LIN {X 0,Y 432.326,Z 417.638,A -85,B 0,C 180,E1 -9497.015,E2 -9497.015} C_VEL
LIN {X 0,Y 432.342,Z 417.631,A -85,B 0,C 180,E1 -9499.819,E2 -9499.819} C_VEL
LIN {X 0,Y 432.316,Z 417.633,A -85,B 0,C 180,E1 -9503.023,E2 -9503.023} C_VEL
LIN {X 0,Y 432.36,Z 417.631,A -85,B 0,C 180,E1 -9505.996,E2 -9505.996} C_VEL
LIN {X 0,Y 432.348,Z 417.629,A -85,B 0,C 180,E1 -9509.49,E2 -9509.49} C_VEL
LIN {X 0,Y 432.394,Z 417.624,A -85,B 0,C 180,E1 -9512.928,E2 -9512.928} C_VEL
LIN {X 0,Y 432.373,Z 417.629,A -85,B 0,C 180,E1 -9516.024,E2 -9516.024} C_VEL
LIN {X 0,Y 432.352,Z 417.628,A -85,B 0,C 180,E1 -9519.046,E2 -9519.046} C_VEL
LIN {X 0,Y 432.38,Z 417.629,A -85,B 0,C 180,E1 -9522.011,E2 -9522.011} C_VEL
LIN {X 0,Y 432.397,Z 417.623,A -85,B 0,C 180,E1 -9524.927,E2 -9524.927} C_VEL
LIN {X 0,Y 432.482,Z 417.615,A -85,B 0,C 180,E1 -9527.804,E2 -9527.804} C_VEL
LIN {X 0,Y 432.465,Z 417.616,A -85,B 0,C 180,E1 -9531.59,E2 -9531.59} C_VEL
LIN {X 0,Y 432.598,Z 417.601,A -85,B 0,C 180,E1 -9534.406,E2 -9534.406} C_VEL
LIN {X 0,Y 432.609,Z 417.6,A -85,B 0,C 180,E1 -9538.138,E2 -9538.138} C_VEL
LIN {X 0,Y 432.735,Z 417.584,A -85,B 0,C 180,E1 -9540,E2 -9540} C_VEL
LIN {X 0,Y 432.594,Z 417.598,A -85,B 0,C 180,E1 -9542.794,E2 -9542.794} C_VEL
LIN {X 0,Y 432.575,Z 417.602,A -85,B 0,C 180,E1 -9546.53,E2 -9546.53} C_VEL
LIN {X 0,Y 432.445,Z 417.618,A -85,B 0,C 180,E1 -9549.353,E2 -9549.353} C_VEL
LIN {X 0,Y 432.432,Z 417.618,A -85,B 0,C 180,E1 -9552.804,E2 -9552.804} C_VEL
LIN {X 0,Y 432.414,Z 417.622,A -85,B 0,C 180,E1 -9556.479,E2 -9556.479} C_VEL
LIN {X 0,Y 432.341,Z 417.633,A -85,B 0,C 180,E1 -9559.961,E2 -9559.961} C_VEL
LIN {X 0,Y 432.322,Z 417.632,A -85,B 0,C 180,E1 -9562.964,E2 -9562.964} C_VEL
LIN {X 0,Y 432.367,Z 417.631,A -85,B 0,C 180,E1 -9566.033,E2 -9566.033} C_VEL
LIN {X 0,Y 432.345,Z 417.629,A -85,B 0,C 180,E1 -9569.188,E2 -9569.188} C_VEL
LIN {X 0,Y 432.325,Z 417.633,A -85,B 0,C 180,E1 -9572.443,E2 -9572.443} C_VEL
LIN {X 0,Y 432.348,Z 417.632,A -85,B 0,C 180,E1 -9575.632,E2 -9575.632} C_VEL
LIN {X 0,Y 432.353,Z 417.628,A -85,B 0,C 180,E1 -9578.716,E2 -9578.716} C_VEL
LIN {X 0,Y 432.338,Z 417.634,A -85,B 0,C 180,E1 -9581.797,E2 -9581.797} C_VEL
LIN {X 0,Y 432.344,Z 417.631,A -85,B 0,C 180,E1 -9584.347,E2 -9584.347} C_VEL
LIN {X 0,Y 432.327,Z 417.632,A -85,B 0,C 180,E1 -9587.015,E2 -9587.015} C_VEL
LIN {X 0,Y 432.34,Z 417.634,A -85,B 0,C 180,E1 -9589.82,E2 -9589.82} C_VEL
LIN {X 0,Y 432.318,Z 417.632,A -85,B 0,C 180,E1 -9593.023,E2 -9593.023} C_VEL
LIN {X 0,Y 432.363,Z 417.63,A -85,B 0,C 180,E1 -9595.997,E2 -9595.997} C_VEL
LIN {X 0,Y 432.399,Z 417.627,A -85,B 0,C 180,E1 -9599.744,E2 -9599.744} C_VEL
LIN {X 0,Y 432.403,Z 417.625,A -85,B 0,C 180,E1 -9603.373,E2 -9603.373} C_VEL
LIN {X 0,Y 432.375,Z 417.629,A -85,B 0,C 180,E1 -9606.024,E2 -9606.024} C_VEL
LIN {X 0,Y 432.355,Z 417.629,A -85,B 0,C 180,E1 -9609.046,E2 -9609.046} C_VEL
LIN {X 0,Y 432.383,Z 417.627,A -85,B 0,C 180,E1 -9612.012,E2 -9612.012} C_VEL
LIN {X 0,Y 432.4,Z 417.626,A -85,B 0,C 180,E1 -9614.927,E2 -9614.927} C_VEL
LIN {X 0,Y 432.461,Z 417.618,A -85,B 0,C 180,E1 -9617.298,E2 -9617.298} C_VEL
LIN {X 0,Y 435.852,Z 429.523,A -85,B 0,C 180,E1 -9618.136,E2 -9618.136} C_VEL
LIN {X 0,Y 436.011,Z 434.479,A -85,B 0,C 180,E1 -9618.494,E2 -9618.494} C_VEL
LIN {X 0,Y 435.45,Z 445.701,A -85,B 0,C 180,E1 -9619.421,E2 -9619.421} C_VEL
LIN {X 0,Y 434.899,Z 455.604,A -85,B 0,C 180,E1 -9620.443,E2 -9620.443} C_VEL
LIN {X 0,Y 434.294,Z 464.879,A -85,B 0,C 180,E1 -9621.626,E2 -9621.626} C_VEL
LIN {X 0,Y 433.884,Z 472.323,A -85,B 0,C 180,E1 -9622.789,E2 -9622.789} C_VEL
LIN {X 0,Y 433.303,Z 479.637,A -85,B 0,C 180,E1 -9624.182,E2 -9624.182} C_VEL
LIN {X 0,Y 432.923,Z 486.364,A -85,B 0,C 180,E1 -9625.811,E2 -9625.811} C_VEL
LIN {X 0,Y 432.607,Z 490.816,A -85,B 0,C 180,E1 -9627.207,E2 -9627.207} C_VEL
LIN {X 0,Y 432.426,Z 493.173,A -85,B 0,C 180,E1 -9628.137,E2 -9628.137} C_VEL
LIN {X 0,Y 432.278,Z 495.194,A -85,B 0,C 180,E1 -9629.127,E2 -9629.127} C_VEL
LIN {X 0,Y 431.525,Z 496.567,A -85,B 0,C 180,E1 -9629.886,E2 -9629.886} C_VEL
LIN {X 0,Y 428.553,Z 498.42,A -85,B 0,C 180,E1 -9631.124,E2 -9631.124} C_VEL
LIN {X 0,Y 426.098,Z 499.436,A -85,B 0,C 180,E1 -9632.129,E2 -9632.129} C_VEL
LIN {X 0,Y 425.064,Z 499.796,A -85,B 0,C 180,E1 -9632.912,E2 -9632.912} C_VEL
LIN {X 0,Y 424.99,Z 499.775,A -85,B 0,C 180,E1 -9633.178,E2 -9633.178} C_VEL
LIN {X 0,Y 425.121,Z 499.284,A -85,B 0,C 180,E1 -9634.742,E2 -9634.742} C_VEL
LIN {X 0,Y 425.3,Z 498.41,A -85,B 0,C 180,E1 -9635.69,E2 -9635.69} C_VEL
LIN {X 0,Y 425.523,Z 495.542,A -85,B 0,C 180,E1 -9637.593,E2 -9637.593} C_VEL
LIN {X 0,Y 425.742,Z 492.253,A -85,B 0,C 180,E1 -9639.023,E2 -9639.023} C_VEL
LIN {X 0,Y 426.172,Z 487.884,A -85,B 0,C 180,E1 -9640.452,E2 -9640.452} C_VEL
LIN {X 0,Y 426.636,Z 481.246,A -85,B 0,C 180,E1 -9642.124,E2 -9642.124} C_VEL
LIN {X 0,Y 427.098,Z 474.255,A -85,B 0,C 180,E1 -9643.516,E2 -9643.516} C_VEL
LIN {X 0,Y 427.766,Z 466.574,A -85,B 0,C 180,E1 -9644.754,E2 -9644.754} C_VEL
LIN {X 0,Y 428.351,Z 457.555,A -85,B 0,C 180,E1 -9645.952,E2 -9645.952} C_VEL
LIN {X 0,Y 428.959,Z 447.467,A -85,B 0,C 180,E1 -9647.03,E2 -9647.03} C_VEL
LIN {X 0,Y 429.566,Z 436.106,A -85,B 0,C 180,E1 -9647.997,E2 -9647.997} C_VEL
LIN {X 0,Y 429.681,Z 432.769,A -85,B 0,C 180,E1 -9648.241,E2 -9648.241} C_VEL
LIN {X 0,Y 426.289,Z 421.626,A -85,B 0,C 180,E1 -9649.115,E2 -9649.115} C_VEL
LIN {X 0,Y 425.389,Z 418.497,A -85,B 0,C 180,E1 -9649.35,E2 -9649.35} C_VEL
LIN {X 0,Y 425.292,Z 418.512,A -85,B 0,C 180,E1 -9652.339,E2 -9652.339} C_VEL
LIN {X 0,Y 425.295,Z 418.504,A -85,B 0,C 180,E1 -9655.446,E2 -9655.446} C_VEL
LIN {X 0,Y 425.353,Z 418.497,A -85,B 0,C 180,E1 -9657.558,E2 -9657.558} C_VEL
LIN {X 0,Y 425.292,Z 418.506,A -85,B 0,C 180,E1 -9660.816,E2 -9660.816} C_VEL
LIN {X 0,Y 425.317,Z 418.508,A -85,B 0,C 180,E1 -9664.288,E2 -9664.288} C_VEL
LIN {X 0,Y 425.284,Z 418.508,A -85,B 0,C 180,E1 -9667.694,E2 -9667.694} C_VEL
LIN {X 0,Y 425.284,Z 418.508,A -85,B 0,C 180,E1 -9670.52,E2 -9670.52} C_VEL
LIN {X 0,Y 425.262,Z 418.509,A -85,B 0,C 180,E1 -9673.351,E2 -9673.351} C_VEL
LIN {X 0,Y 425.263,Z 418.509,A -85,B 0,C 180,E1 -9676.649,E2 -9676.649} C_VEL
LIN {X 0,Y 425.291,Z 418.51,A -85,B 0,C 180,E1 -9679.873,E2 -9679.873} C_VEL
LIN {X 0,Y 425.282,Z 418.508,A -85,B 0,C 180,E1 -9682.488,E2 -9682.488} C_VEL
LIN {X 0,Y 425.312,Z 418.508,A -85,B 0,C 180,E1 -9685.817,E2 -9685.817} C_VEL
LIN {X 0,Y 425.295,Z 418.505,A -85,B 0,C 180,E1 -9689.239,E2 -9689.239} C_VEL
LIN {X 0,Y 425.353,Z 418.498,A -85,B 0,C 180,E1 -9692.442,E2 -9692.442} C_VEL
LIN {X 0,Y 425.352,Z 418.502,A -85,B 0,C 180,E1 -9695.602,E2 -9695.602} C_VEL
LIN {X 0,Y 425.297,Z 418.504,A -85,B 0,C 180,E1 -9698.681,E2 -9698.681} C_VEL
LIN {X 0,Y 425.334,Z 418.507,A -85,B 0,C 180,E1 -9701.703,E2 -9701.703} C_VEL
LIN {X 0,Y 425.352,Z 418.497,A -85,B 0,C 180,E1 -9704.671,E2 -9704.671} C_VEL
LIN {X 0,Y 425.39,Z 418.497,A -85,B 0,C 180,E1 -9705.468,E2 -9705.468} C_VEL
LIN {X 0,Y 428.481,Z 430.294,A -85,B 0,C 180,E1 -9706.336,E2 -9706.336} C_VEL
LIN {X 0,Y 428.042,Z 441.217,A -85,B 0,C 180,E1 -9707.193,E2 -9707.193} C_VEL
LIN {X 0,Y 427.389,Z 452.229,A -85,B 0,C 180,E1 -9708.258,E2 -9708.258} C_VEL
LIN {X 0,Y 427.073,Z 461.189,A -85,B 0,C 180,E1 -9709.331,E2 -9709.331} C_VEL
LIN {X 0,Y 426.483,Z 470.942,A -85,B 0,C 180,E1 -9710.754,E2 -9710.754} C_VEL
LIN {X 0,Y 426.118,Z 478.16,A -85,B 0,C 180,E1 -9712.05,E2 -9712.05} C_VEL
LIN {X 0,Y 425.716,Z 484.179,A -85,B 0,C 180,E1 -9713.364,E2 -9713.364} C_VEL
LIN {X 0,Y 425.501,Z 489.404,A -85,B 0,C 180,E1 -9714.788,E2 -9714.788} C_VEL
LIN {X 0,Y 425.181,Z 493.494,A -85,B 0,C 180,E1 -9716.209,E2 -9716.209} C_VEL
LIN {X 0,Y 425.043,Z 495.618,A -85,B 0,C 180,E1 -9717.157,E2 -9717.157} C_VEL
LIN {X 0,Y 425.115,Z 497.314,A -85,B 0,C 180,E1 -9718.105,E2 -9718.105} C_VEL
LIN {X 0,Y 425.026,Z 498.601,A -85,B 0,C 180,E1 -9719.052,E2 -9719.052} C_VEL
LIN {X 0,Y 425.094,Z 499.904,A -85,B 0,C 180,E1 -9720.947,E2 -9720.947} C_VEL
LIN {X 0,Y 425.168,Z 499.97,A -85,B 0,C 180,E1 -9721.894,E2 -9721.894} C_VEL
LIN {X 0,Y 425.207,Z 498.846,A -85,B 0,C 180,E1 -9723.791,E2 -9723.791} C_VEL
LIN {X 0,Y 425.335,Z 497.69,A -85,B 0,C 180,E1 -9724.739,E2 -9724.739} C_VEL
LIN {X 0,Y 425.688,Z 495.116,A -85,B 0,C 180,E1 -9726.16,E2 -9726.16} C_VEL
LIN {X 0,Y 426.087,Z 490.636,A -85,B 0,C 180,E1 -9727.877,E2 -9727.877} C_VEL
LIN {X 0,Y 426.537,Z 484.964,A -85,B 0,C 180,E1 -9729.484,E2 -9729.484} C_VEL
LIN {X 0,Y 427.038,Z 478.492,A -85,B 0,C 180,E1 -9730.91,E2 -9730.91} C_VEL
LIN {X 0,Y 427.718,Z 470.343,A -85,B 0,C 180,E1 -9732.334,E2 -9732.334} C_VEL
LIN {X 0,Y 428.268,Z 462.012,A -85,B 0,C 180,E1 -9733.524,E2 -9733.524} C_VEL
LIN {X 0,Y 428.866,Z 452.834,A -85,B 0,C 180,E1 -9734.601,E2 -9734.601} C_VEL
LIN {X 0,Y 429.587,Z 441.586,A -85,B 0,C 180,E1 -9735.661,E2 -9735.661} C_VEL
LIN {X 0,Y 429.924,Z 432.512,A -85,B 0,C 180,E1 -9736.362,E2 -9736.362} C_VEL
LIN {X 0,Y 426.422,Z 421.828,A -85,B 0,C 180,E1 -9737.257,E2 -9737.257} C_VEL
LIN {X 0,Y 425.383,Z 418.504,A -85,B 0,C 180,E1 -9737.518,E2 -9737.518} C_VEL
LIN {X 0,Y 425.299,Z 418.517,A -85,B 0,C 180,E1 -9740.305,E2 -9740.305} C_VEL
LIN {X 0,Y 425.308,Z 418.51,A -85,B 0,C 180,E1 -9743.365,E2 -9743.365} C_VEL
LIN {X 0,Y 425.351,Z 418.503,A -85,B 0,C 180,E1 -9746.844,E2 -9746.844} C_VEL
LIN {X 0,Y 425.294,Z 418.509,A -85,B 0,C 180,E1 -9749.719,E2 -9749.719} C_VEL
LIN {X 0,Y 425.285,Z 418.51,A -85,B 0,C 180,E1 -9753.048,E2 -9753.048} C_VEL
LIN {X 0,Y 425.285,Z 418.511,A -85,B 0,C 180,E1 -9755.928,E2 -9755.928} C_VEL
LIN {X 0,Y 425.296,Z 418.508,A -85,B 0,C 180,E1 -9759.042,E2 -9759.042} C_VEL
LIN {X 0,Y 425.278,Z 418.513,A -85,B 0,C 180,E1 -9762.653,E2 -9762.653} C_VEL
LIN {X 0,Y 425.264,Z 418.51,A -85,B 0,C 180,E1 -9766.044,E2 -9766.044} C_VEL
LIN {X 0,Y 425.364,Z 418.669,A -85,B 0,C 180,E1 -9767.585,E2 -9767.585} C_VEL
LIN {X 0,Y 427.208,Z 427.813,A -85,B 0,C 180,E1 -9770.642,E2 -9770.642} C_VEL
LIN {X 0,Y 428.572,Z 435.789,A -85,B 0,C 180,E1 -9773.117,E2 -9773.117} C_VEL
LIN {X 0,Y 427.809,Z 446.144,A -85,B 0,C 180,E1 -9776.044,E2 -9776.044} C_VEL
LIN {X 0,Y 427.039,Z 458.13,A -85,B 0,C 180,E1 -9779.324,E2 -9779.324} C_VEL
LIN {X 0,Y 426.387,Z 470.133,A -85,B 0,C 180,E1 -9782.515,E2 -9782.515} C_VEL
LIN {X 0,Y 425.854,Z 482.082,A -85,B 0,C 180,E1 -9785.633,E2 -9785.633} C_VEL
LIN {X 0,Y 425.349,Z 493.918,A -85,B 0,C 180,E1 -9788.684,E2 -9788.684} C_VEL
LIN {X 0,Y 425.005,Z 505.578,A -85,B 0,C 180,E1 -9791.688,E2 -9791.688} C_VEL
LIN {X 0,Y 424.9,Z 510.092,A -85,B 0,C 180,E1 -9792.85,E2 -9792.85} C_VEL
LIN {X 0,Y 426.68,Z 525.47,A -85,B 0,C 180,E1 -9793.351,E2 -9793.351} C_VEL
LIN {X 0,Y 427.444,Z 538.57,A -85,B 0,C 180,E1 -9793.952,E2 -9793.952} C_VEL
LIN {X 0,Y 427.871,Z 548.142,A -85,B 0,C 180,E1 -9794.519,E2 -9794.519} C_VEL
LIN {X 0,Y 427.109,Z 559.694,A -85,B 0,C 180,E1 -9795.345,E2 -9795.345} C_VEL
LIN {X 0,Y 426.337,Z 571.448,A -85,B 0,C 180,E1 -9796.414,E2 -9796.414} C_VEL
LIN {X 0,Y 425.858,Z 580.24,A -85,B 0,C 180,E1 -9797.401,E2 -9797.401} C_VEL
LIN {X 0,Y 425.303,Z 588.867,A -85,B 0,C 180,E1 -9798.562,E2 -9798.562} C_VEL
LIN {X 0,Y 424.829,Z 597.558,A -85,B 0,C 180,E1 -9799.997,E2 -9799.997} C_VEL
LIN {X 0,Y 424.634,Z 604.578,A -85,B 0,C 180,E1 -9801.433,E2 -9801.433} C_VEL
LIN {X 0,Y 424.578,Z 610.395,A -85,B 0,C 180,E1 -9802.916,E2 -9802.916} C_VEL
LIN {X 0,Y 424.589,Z 614.669,A -85,B 0,C 180,E1 -9804.3,E2 -9804.3} C_VEL
LIN {X 0,Y 424.686,Z 617.04,A -85,B 0,C 180,E1 -9805.253,E2 -9805.253} C_VEL
LIN {X 0,Y 424.718,Z 618.941,A -85,B 0,C 180,E1 -9806.205,E2 -9806.205} C_VEL
LIN {X 0,Y 424.7,Z 620.365,A -85,B 0,C 180,E1 -9807.154,E2 -9807.154} C_VEL
LIN {X 0,Y 424.921,Z 622.033,A -85,B 0,C 180,E1 -9809.052,E2 -9809.052} C_VEL
LIN {X 0,Y 424.922,Z 622.232,A -85,B 0,C 180,E1 -9810,E2 -9810} C_VEL
LIN {X 0,Y 424.922,Z 621.99,A -85,B 0,C 180,E1 -9810.947,E2 -9810.947} C_VEL
LIN {X 0,Y 424.71,Z 620.274,A -85,B 0,C 180,E1 -9812.845,E2 -9812.845} C_VEL
LIN {X 0,Y 424.715,Z 618.797,A -85,B 0,C 180,E1 -9813.795,E2 -9813.795} C_VEL
LIN {X 0,Y 424.651,Z 615.717,A -85,B 0,C 180,E1 -9815.222,E2 -9815.222} C_VEL
LIN {X 0,Y 424.582,Z 611.387,A -85,B 0,C 180,E1 -9816.702,E2 -9816.702} C_VEL
LIN {X 0,Y 424.656,Z 605.163,A -85,B 0,C 180,E1 -9818.326,E2 -9818.326} C_VEL
LIN {X 0,Y 424.83,Z 598.22,A -85,B 0,C 180,E1 -9819.762,E2 -9819.762} C_VEL
LIN {X 0,Y 425.196,Z 589.631,A -85,B 0,C 180,E1 -9821.199,E2 -9821.199} C_VEL
LIN {X 0,Y 425.761,Z 580.824,A -85,B 0,C 180,E1 -9822.391,E2 -9822.391} C_VEL
LIN {X 0,Y 426.226,Z 571.171,A -85,B 0,C 180,E1 -9823.468,E2 -9823.468} C_VEL
LIN {X 0,Y 426.938,Z 559.25,A -85,B 0,C 180,E1 -9824.539,E2 -9824.539} C_VEL
LIN {X 0,Y 427.689,Z 547.375,A -85,B 0,C 180,E1 -9825.365,E2 -9825.365} C_VEL
LIN {X 0,Y 427.38,Z 540.977,A -85,B 0,C 180,E1 -9825.743,E2 -9825.743} C_VEL
LIN {X 0,Y 426.502,Z 527.164,A -85,B 0,C 180,E1 -9826.399,E2 -9826.399} C_VEL
LIN {X 0,Y 425.159,Z 513.732,A -85,B 0,C 180,E1 -9826.84,E2 -9826.84} C_VEL
LIN {X 0,Y 424.856,Z 510.351,A -85,B 0,C 180,E1 -9826.941,E2 -9826.941} C_VEL
LIN {X 0,Y 425.219,Z 497.119,A -85,B 0,C 180,E1 -9830.309,E2 -9830.309} C_VEL
LIN {X 0,Y 425.617,Z 485.211,A -85,B 0,C 180,E1 -9833.347,E2 -9833.347} C_VEL
LIN {X 0,Y 426.117,Z 473.121,A -85,B 0,C 180,E1 -9836.443,E2 -9836.443} C_VEL
LIN {X 0,Y 426.832,Z 458.896,A -85,B 0,C 180,E1 -9840.145,E2 -9840.145} C_VEL
LIN {X 0,Y 427.475,Z 446.582,A -85,B 0,C 180,E1 -9843.438,E2 -9843.438} C_VEL
LIN {X 0,Y 428.244,Z 435.561,A -85,B 0,C 180,E1 -9846.472,E2 -9846.472} C_VEL
LIN {X 0,Y 427.7,Z 430.625,A -85,B 0,C 180,E1 -9847.932,E2 -9847.932} C_VEL
LIN {X 0,Y 425.77,Z 420.667,A -85,B 0,C 180,E1 -9851.058,E2 -9851.058} C_VEL
LIN {X 0,Y 425.335,Z 418.505,A -85,B 0,C 180,E1 -9851.768,E2 -9851.768} C_VEL
LIN {X 0,Y 425.29,Z 418.513,A -85,B 0,C 180,E1 -9855.282,E2 -9855.282} C_VEL
LIN {X 0,Y 425.277,Z 418.512,A -85,B 0,C 180,E1 -9858.622,E2 -9858.622} C_VEL
LIN {X 0,Y 425.317,Z 418.505,A -85,B 0,C 180,E1 -9861.103,E2 -9861.103} C_VEL
LIN {X 0,Y 425.301,Z 418.508,A -85,B 0,C 180,E1 -9864.664,E2 -9864.664} C_VEL
LIN {X 0,Y 425.266,Z 418.515,A -85,B 0,C 180,E1 -9868.073,E2 -9868.073} C_VEL
LIN {X 0,Y 425.332,Z 418.503,A -85,B 0,C 180,E1 -9871.368,E2 -9871.368} C_VEL
LIN {X 0,Y 425.297,Z 418.509,A -85,B 0,C 180,E1 -9874.555,E2 -9874.555} C_VEL
LIN {X 0,Y 425.289,Z 418.51,A -85,B 0,C 180,E1 -9877.661,E2 -9877.661} C_VEL
LIN {X 0,Y 425.363,Z 418.5,A -85,B 0,C 180,E1 -9880.704,E2 -9880.704} C_VEL
LIN {X 0,Y 425.39,Z 418.497,A -85,B 0,C 180,E1 -9883.688,E2 -9883.688} C_VEL
LIN {X 0,Y 425.431,Z 418.492,A -85,B 0,C 180,E1 -9887.599,E2 -9887.599} C_VEL
LIN {X 0,Y 425.41,Z 418.493,A -85,B 0,C 180,E1 -9891.449,E2 -9891.449} C_VEL
LIN {X 0,Y 425.554,Z 418.479,A -85,B 0,C 180,E1 -9894.313,E2 -9894.313} C_VEL
LIN {X 0,Y 425.578,Z 418.476,A -85,B 0,C 180,E1 -9898.107,E2 -9898.107} C_VEL
LIN {X 0,Y 425.705,Z 418.46,A -85,B 0,C 180,E1 -9900,E2 -9900} C_VEL
LIN {X 0,Y 425.547,Z 418.475,A -85,B 0,C 180,E1 -9902.84,E2 -9902.84} C_VEL
LIN {X 0,Y 425.532,Z 418.478,A -85,B 0,C 180,E1 -9906.649,E2 -9906.649} C_VEL
LIN {X 0,Y 425.403,Z 418.496,A -85,B 0,C 180,E1 -9909.51,E2 -9909.51} C_VEL
LIN {X 0,Y 425.395,Z 418.495,A -85,B 0,C 180,E1 -9912.904,E2 -9912.904} C_VEL
LIN {X 0,Y 425.363,Z 418.499,A -85,B 0,C 180,E1 -9916.605,E2 -9916.605} C_VEL
LIN {X 0,Y 425.331,Z 418.505,A -85,B 0,C 180,E1 -9919.636,E2 -9919.636} C_VEL
LIN {X 0,Y 425.309,Z 418.507,A -85,B 0,C 180,E1 -9923.365,E2 -9923.365} C_VEL
LIN {X 0,Y 425.35,Z 418.5,A -85,B 0,C 180,E1 -9926.845,E2 -9926.845} C_VEL
LIN {X 0,Y 425.293,Z 418.512,A -85,B 0,C 180,E1 -9929.72,E2 -9929.72} C_VEL
LIN {X 0,Y 425.284,Z 418.509,A -85,B 0,C 180,E1 -9933.048,E2 -9933.048} C_VEL
LIN {X 0,Y 425.287,Z 418.513,A -85,B 0,C 180,E1 -9935.929,E2 -9935.929} C_VEL
LIN {X 0,Y 425.302,Z 418.506,A -85,B 0,C 180,E1 -9939.044,E2 -9939.044} C_VEL
LIN {X 0,Y 425.28,Z 418.509,A -85,B 0,C 180,E1 -9942.653,E2 -9942.653} C_VEL
LIN {X 0,Y 425.271,Z 418.513,A -85,B 0,C 180,E1 -9946.045,E2 -9946.045} C_VEL
LIN {X 0,Y 425.278,Z 418.509,A -85,B 0,C 180,E1 -9948.622,E2 -9948.622} C_VEL
LIN {X 0,Y 425.316,Z 418.505,A -85,B 0,C 180,E1 -9951.103,E2 -9951.103} C_VEL
LIN {X 0,Y 425.303,Z 418.506,A -85,B 0,C 180,E1 -9954.665,E2 -9954.665} C_VEL
LIN {X 0,Y 425.276,Z 418.513,A -85,B 0,C 180,E1 -9958.074,E2 -9958.074} C_VEL
LIN {X 0,Y 425.341,Z 418.505,A -85,B 0,C 180,E1 -9961.369,E2 -9961.369} C_VEL
LIN {X 0,Y 425.299,Z 418.506,A -85,B 0,C 180,E1 -9964.555,E2 -9964.555} C_VEL
LIN {X 0,Y 425.291,Z 418.512,A -85,B 0,C 180,E1 -9967.662,E2 -9967.662} C_VEL
LIN {X 0,Y 425.366,Z 418.498,A -85,B 0,C 180,E1 -9970.704,E2 -9970.704} C_VEL
LIN {X 0,Y 425.393,Z 418.499,A -85,B 0,C 180,E1 -9973.689,E2 -9973.689} C_VEL
LIN {X 0,Y 425.401,Z 418.497,A -85,B 0,C 180,E1 -9977.032,E2 -9977.032} C_VEL
LIN {X 0,Y 429.015,Z 431.02,A -85,B 0,C 180,E1 -9977.944,E2 -9977.944} C_VEL
LIN {X 0,Y 429.174,Z 435.923,A -85,B 0,C 180,E1 -9978.308,E2 -9978.308} C_VEL
LIN {X 0,Y 428.604,Z 447.061,A -85,B 0,C 180,E1 -9979.25,E2 -9979.25} C_VEL
LIN {X 0,Y 428.016,Z 456.896,A -85,B 0,C 180,E1 -9980.287,E2 -9980.287} C_VEL
LIN {X 0,Y 427.377,Z 466.112,A -85,B 0,C 180,E1 -9981.489,E2 -9981.489} C_VEL
LIN {X 0,Y 426.942,Z 473.519,A -85,B 0,C 180,E1 -9982.671,E2 -9982.671} C_VEL
LIN {X 0,Y 426.338,Z 480.801,A -85,B 0,C 180,E1 -9984.087,E2 -9984.087} C_VEL
LIN {X 0,Y 425.934,Z 487.494,A -85,B 0,C 180,E1 -9985.742,E2 -9985.742} C_VEL
LIN {X 0,Y 425.603,Z 491.92,A -85,B 0,C 180,E1 -9987.161,E2 -9987.161} C_VEL
LIN {X 0,Y 425.417,Z 494.257,A -85,B 0,C 180,E1 -9988.107,E2 -9988.107} C_VEL
LIN {X 0,Y 425.194,Z 497.682,A -85,B 0,C 180,E1 -9990,E2 -9990} C_VEL
LIN {X 0,Y 425.026,Z 498.79,A -85,B 0,C 180,E1 -9990.948,E2 -9990.948} C_VEL
LIN {X 0,Y 425.097,Z 499.462,A -85,B 0,C 180,E1 -9991.895,E2 -9991.895} C_VEL
LIN {X 0,Y 424.99,Z 499.775,A -85,B 0,C 180,E1 -9993.178,E2 -9993.178} C_VEL
LIN {X 0,Y 424.374,Z 499.785,A -85,B 0,C 180,E1 -9993.971,E2 -9993.971} C_VEL
LIN {X 0,Y 421.648,Z 499.39,A -85,B 0,C 180,E1 -9995.263,E2 -9995.263} C_VEL
LIN {X 0,Y 418.977,Z 498.335,A -85,B 0,C 180,E1 -9996.561,E2 -9996.561} C_VEL
LIN {X 0,Y 418.459,Z 497.119,A -85,B 0,C 180,E1 -9997.353,E2 -9997.353} C_VEL
LIN {X 0,Y 418.795,Z 493.18,A -85,B 0,C 180,E1 -9999.174,E2 -9999.174} C_VEL
LIN {X 0,Y 419.251,Z 488.785,A -85,B 0,C 180,E1 -10000.626,E2 -10000.626} C_VEL
LIN {X 0,Y 419.738,Z 482.107,A -85,B 0,C 180,E1 -10002.327,E2 -10002.327} C_VEL
LIN {X 0,Y 420.243,Z 475.129,A -85,B 0,C 180,E1 -10003.732,E2 -10003.732} C_VEL
LIN {X 0,Y 420.959,Z 467.363,A -85,B 0,C 180,E1 -10004.998,E2 -10004.998} C_VEL
LIN {X 0,Y 421.552,Z 458.292,A -85,B 0,C 180,E1 -10006.216,E2 -10006.216} C_VEL
LIN {X 0,Y 422.205,Z 448.128,A -85,B 0,C 180,E1 -10007.311,E2 -10007.311} C_VEL
LIN {X 0,Y 422.843,Z 436.401,A -85,B 0,C 180,E1 -10008.316,E2 -10008.316} C_VEL
LIN {X 0,Y 422.588,Z 433.25,A -85,B 0,C 180,E1 -10008.564,E2 -10008.564} C_VEL
LIN {X 0,Y 419.259,Z 422.462,A -85,B 0,C 180,E1 -10009.425,E2 -10009.425} C_VEL
LIN {X 0,Y 418.312,Z 419.38,A -85,B 0,C 180,E1 -10009.671,E2 -10009.671} C_VEL
LIN {X 0,Y 418.236,Z 419.386,A -85,B 0,C 180,E1 -10012.737,E2 -10012.737} C_VEL
LIN {X 0,Y 418.272,Z 419.382,A -85,B 0,C 180,E1 -10015.904,E2 -10015.904} C_VEL
LIN {X 0,Y 418.269,Z 419.379,A -85,B 0,C 180,E1 -10019.162,E2 -10019.162} C_VEL
LIN {X 0,Y 418.262,Z 419.381,A -85,B 0,C 180,E1 -10022.844,E2 -10022.844} C_VEL
LIN {X 0,Y 418.25,Z 419.389,A -85,B 0,C 180,E1 -10026.238,E2 -10026.238} C_VEL
LIN {X 0,Y 418.253,Z 419.384,A -85,B 0,C 180,E1 -10029.682,E2 -10029.682} C_VEL
LIN {X 0,Y 418.234,Z 419.388,A -85,B 0,C 180,E1 -10032.321,E2 -10032.321} C_VEL
LIN {X 0,Y 418.242,Z 419.383,A -85,B 0,C 180,E1 -10035.109,E2 -10035.109} C_VEL
LIN {X 0,Y 418.245,Z 419.387,A -85,B 0,C 180,E1 -10037.767,E2 -10037.767} C_VEL
LIN {X 0,Y 418.257,Z 419.382,A -85,B 0,C 180,E1 -10040.619,E2 -10040.619} C_VEL
LIN {X 0,Y 418.248,Z 419.389,A -85,B 0,C 180,E1 -10043.976,E2 -10043.976} C_VEL
LIN {X 0,Y 418.262,Z 419.381,A -85,B 0,C 180,E1 -10047.156,E2 -10047.156} C_VEL
LIN {X 0,Y 418.273,Z 419.379,A -85,B 0,C 180,E1 -10050.895,E2 -10050.895} C_VEL
LIN {X 0,Y 418.272,Z 419.383,A -85,B 0,C 180,E1 -10054.096,E2 -10054.096} C_VEL
LIN {X 0,Y 418.236,Z 419.385,A -85,B 0,C 180,E1 -10057.263,E2 -10057.263} C_VEL
LIN {X 0,Y 418.287,Z 419.378,A -85,B 0,C 180,E1 -10060.364,E2 -10060.364} C_VEL
LIN {X 0,Y 418.321,Z 419.377,A -85,B 0,C 180,E1 -10063.405,E2 -10063.405} C_VEL
LIN {X 0,Y 418.352,Z 419.469,A -85,B 0,C 180,E1 -10065.28,E2 -10065.28} C_VEL
LIN {X 0,Y 421.505,Z 431.457,A -85,B 0,C 180,E1 -10066.168,E2 -10066.168} C_VEL
LIN {X 0,Y 421.057,Z 443.001,A -85,B 0,C 180,E1 -10067.1,E2 -10067.1} C_VEL
LIN {X 0,Y 420.413,Z 453.841,A -85,B 0,C 180,E1 -10068.183,E2 -10068.183} C_VEL
LIN {X 0,Y 420.022,Z 463.566,A -85,B 0,C 180,E1 -10069.394,E2 -10069.394} C_VEL
LIN {X 0,Y 419.45,Z 473.098,A -85,B 0,C 180,E1 -10070.841,E2 -10070.841} C_VEL
LIN {X 0,Y 419.033,Z 480.704,A -85,B 0,C 180,E1 -10072.289,E2 -10072.289} C_VEL
LIN {X 0,Y 418.636,Z 486.865,A -85,B 0,C 180,E1 -10073.735,E2 -10073.735} C_VEL
LIN {X 0,Y 418.281,Z 491.774,A -85,B 0,C 180,E1 -10075.181,E2 -10075.181} C_VEL
LIN {X 0,Y 418.176,Z 495.538,A -85,B 0,C 180,E1 -10076.628,E2 -10076.628} C_VEL
LIN {X 0,Y 418.093,Z 498.285,A -85,B 0,C 180,E1 -10078.073,E2 -10078.073} C_VEL
LIN {X 0,Y 418.004,Z 499.603,A -85,B 0,C 180,E1 -10079.036,E2 -10079.036} C_VEL
LIN {X 0,Y 418.092,Z 500.947,A -85,B 0,C 180,E1 -10080.963,E2 -10080.963} C_VEL
LIN {X 0,Y 418.172,Z 501.042,A -85,B 0,C 180,E1 -10081.926,E2 -10081.926} C_VEL
LIN {X 0,Y 418.183,Z 500.705,A -85,B 0,C 180,E1 -10082.89,E2 -10082.89} C_VEL
LIN {X 0,Y 418.352,Z 498.848,A -85,B 0,C 180,E1 -10084.818,E2 -10084.818} C_VEL
LIN {X 0,Y 418.74,Z 496.304,A -85,B 0,C 180,E1 -10086.263,E2 -10086.263} C_VEL
LIN {X 0,Y 419.103,Z 492.756,A -85,B 0,C 180,E1 -10087.71,E2 -10087.71} C_VEL
LIN {X 0,Y 419.482,Z 488.079,A -85,B 0,C 180,E1 -10089.158,E2 -10089.158} C_VEL
LIN {X 0,Y 420.046,Z 480.96,A -85,B 0,C 180,E1 -10090.849,E2 -10090.849} C_VEL
LIN {X 0,Y 420.742,Z 473.242,A -85,B 0,C 180,E1 -10092.297,E2 -10092.297} C_VEL
LIN {X 0,Y 421.513,Z 463.526,A -85,B 0,C 180,E1 -10093.745,E2 -10093.745} C_VEL
LIN {X 0,Y 422.165,Z 454.459,A -85,B 0,C 180,E1 -10094.838,E2 -10094.838} C_VEL
LIN {X 0,Y 422.944,Z 443.313,A -85,B 0,C 180,E1 -10095.913,E2 -10095.913} C_VEL
LIN {X 0,Y 423.32,Z 434.494,A -85,B 0,C 180,E1 -10096.615,E2 -10096.615} C_VEL
LIN {X 0,Y 419.956,Z 424.093,A -85,B 0,C 180,E1 -10097.532,E2 -10097.532} C_VEL
LIN {X 0,Y 418.32,Z 419.386,A -85,B 0,C 180,E1 -10097.918,E2 -10097.918} C_VEL
LIN {X 0,Y 418.254,Z 419.393,A -85,B 0,C 180,E1 -10100.663,E2 -10100.663} C_VEL
LIN {X 0,Y 418.289,Z 419.384,A -85,B 0,C 180,E1 -10103.781,E2 -10103.781} C_VEL
LIN {X 0,Y 418.313,Z 419.381,A -85,B 0,C 180,E1 -10107.07,E2 -10107.07} C_VEL
LIN {X 0,Y 418.248,Z 419.388,A -85,B 0,C 180,E1 -10110.272,E2 -10110.272} C_VEL
LIN {X 0,Y 418.252,Z 419.384,A -85,B 0,C 180,E1 -10113.677,E2 -10113.677} C_VEL
LIN {X 0,Y 418.243,Z 419.386,A -85,B 0,C 180,E1 -10117.224,E2 -10117.224} C_VEL
LIN {X 0,Y 418.252,Z 419.386,A -85,B 0,C 180,E1 -10119.682,E2 -10119.682} C_VEL
LIN {X 0,Y 418.233,Z 419.387,A -85,B 0,C 180,E1 -10122.321,E2 -10122.321} C_VEL
LIN {X 0,Y 418.239,Z 419.392,A -85,B 0,C 180,E1 -10125.109,E2 -10125.109} C_VEL
LIN {X 0,Y 418.281,Z 419.414,A -85,B 0,C 180,E1 -10127.176,E2 -10127.176} C_VEL
LIN {X 0,Y 420.304,Z 429.337,A -85,B 0,C 180,E1 -10130.549,E2 -10130.549} C_VEL
LIN {X 0,Y 421.572,Z 436.433,A -85,B 0,C 180,E1 -10132.82,E2 -10132.82} C_VEL
LIN {X 0,Y 421.307,Z 441.408,A -85,B 0,C 180,E1 -10134.278,E2 -10134.278} C_VEL
LIN {X 0,Y 420.417,Z 453.36,A -85,B 0,C 180,E1 -10137.66,E2 -10137.66} C_VEL
LIN {X 0,Y 419.68,Z 465.323,A -85,B 0,C 180,E1 -10140.945,E2 -10140.945} C_VEL
LIN {X 0,Y 418.956,Z 478.963,A -85,B 0,C 180,E1 -10144.601,E2 -10144.601} C_VEL
LIN {X 0,Y 418.416,Z 491.422,A -85,B 0,C 180,E1 -10147.891,E2 -10147.891} C_VEL
LIN {X 0,Y 417.955,Z 504.601,A -85,B 0,C 180,E1 -10151.368,E2 -10151.368} C_VEL
LIN {X 0,Y 417.835,Z 509.039,A -85,B 0,C 180,E1 -10152.531,E2 -10152.531} C_VEL
LIN {X 0,Y 419.633,Z 524.36,A -85,B 0,C 180,E1 -10153.042,E2 -10153.042} C_VEL
LIN {X 0,Y 420.484,Z 537.86,A -85,B 0,C 180,E1 -10153.679,E2 -10153.679} C_VEL
LIN {X 0,Y 420.982,Z 547.376,A -85,B 0,C 180,E1 -10154.259,E2 -10154.259} C_VEL
LIN {X 0,Y 420.198,Z 558.868,A -85,B 0,C 180,E1 -10155.099,E2 -10155.099} C_VEL
LIN {X 0,Y 419.378,Z 570.578,A -85,B 0,C 180,E1 -10156.184,E2 -10156.184} C_VEL
LIN {X 0,Y 418.841,Z 579.616,A -85,B 0,C 180,E1 -10157.221,E2 -10157.221} C_VEL
LIN {X 0,Y 418.27,Z 587.945,A -85,B 0,C 180,E1 -10158.367,E2 -10158.367} C_VEL
LIN {X 0,Y 417.762,Z 596.607,A -85,B 0,C 180,E1 -10159.826,E2 -10159.826} C_VEL
LIN {X 0,Y 417.558,Z 603.614,A -85,B 0,C 180,E1 -10161.287,E2 -10161.287} C_VEL
LIN {X 0,Y 417.497,Z 609.252,A -85,B 0,C 180,E1 -10162.747,E2 -10162.747} C_VEL
LIN {X 0,Y 417.535,Z 613.688,A -85,B 0,C 180,E1 -10164.203,E2 -10164.203} C_VEL
LIN {X 0,Y 417.638,Z 616.055,A -85,B 0,C 180,E1 -10165.173,E2 -10165.173} C_VEL
LIN {X 0,Y 417.68,Z 617.947,A -85,B 0,C 180,E1 -10166.141,E2 -10166.141} C_VEL
LIN {X 0,Y 417.657,Z 619.366,A -85,B 0,C 180,E1 -10167.106,E2 -10167.106} C_VEL
LIN {X 0,Y 417.897,Z 621.028,A -85,B 0,C 180,E1 -10169.036,E2 -10169.036} C_VEL
LIN {X 0,Y 417.902,Z 621.218,A -85,B 0,C 180,E1 -10170,E2 -10170} C_VEL
LIN {X 0,Y 417.898,Z 620.971,A -85,B 0,C 180,E1 -10170.963,E2 -10170.963} C_VEL
LIN {X 0,Y 417.669,Z 619.241,A -85,B 0,C 180,E1 -10172.893,E2 -10172.893} C_VEL
LIN {X 0,Y 417.677,Z 617.753,A -85,B 0,C 180,E1 -10173.859,E2 -10173.859} C_VEL
LIN {X 0,Y 417.587,Z 614.658,A -85,B 0,C 180,E1 -10175.311,E2 -10175.311} C_VEL
LIN {X 0,Y 417.519,Z 610.476,A -85,B 0,C 180,E1 -10176.767,E2 -10176.767} C_VEL
LIN {X 0,Y 417.586,Z 604.067,A -85,B 0,C 180,E1 -10178.468,E2 -10178.468} C_VEL
LIN {X 0,Y 417.778,Z 597.106,A -85,B 0,C 180,E1 -10179.929,E2 -10179.929} C_VEL
LIN {X 0,Y 418.179,Z 588.492,A -85,B 0,C 180,E1 -10181.389,E2 -10181.389} C_VEL
LIN {X 0,Y 418.793,Z 579.662,A -85,B 0,C 180,E1 -10182.601,E2 -10182.601} C_VEL
LIN {X 0,Y 418.986,Z 573.052,A -85,B 0,C 180,E1 -10183.373,E2 -10183.373} C_VEL
LIN {X 0,Y 419.756,Z 562.354,A -85,B 0,C 180,E1 -10184.421,E2 -10184.421} C_VEL
LIN {X 0,Y 420.462,Z 551.567,A -85,B 0,C 180,E1 -10185.263,E2 -10185.263} C_VEL
LIN {X 0,Y 420.688,Z 545.022,A -85,B 0,C 180,E1 -10185.69,E2 -10185.69} C_VEL
LIN {X 0,Y 419.993,Z 534.664,A -85,B 0,C 180,E1 -10186.277,E2 -10186.277} C_VEL
LIN {X 0,Y 419.012,Z 521.336,A -85,B 0,C 180,E1 -10186.844,E2 -10186.844} C_VEL
LIN {X 0,Y 417.783,Z 509.362,A -85,B 0,C 180,E1 -10187.205,E2 -10187.205} C_VEL
LIN {X 0,Y 418.158,Z 496.065,A -85,B 0,C 180,E1 -10190.668,E2 -10190.668} C_VEL
LIN {X 0,Y 418.648,Z 483.195,A -85,B 0,C 180,E1 -10194.022,E2 -10194.022} C_VEL
LIN {X 0,Y 419.187,Z 470.681,A -85,B 0,C 180,E1 -10197.304,E2 -10197.304} C_VEL
LIN {X 0,Y 419.895,Z 457.951,A -85,B 0,C 180,E1 -10200.697,E2 -10200.697} C_VEL
LIN {X 0,Y 420.698,Z 444.727,A -85,B 0,C 180,E1 -10204.32,E2 -10204.32} C_VEL
LIN {X 0,Y 421.264,Z 435.571,A -85,B 0,C 180,E1 -10206.912,E2 -10206.912} C_VEL
LIN {X 0,Y 419.784,Z 426.792,A -85,B 0,C 180,E1 -10209.634,E2 -10209.634} C_VEL
LIN {X 0,Y 418.28,Z 419.383,A -85,B 0,C 180,E1 -10212.097,E2 -10212.097} C_VEL
LIN {X 0,Y 418.24,Z 419.392,A -85,B 0,C 180,E1 -10215.109,E2 -10215.109} C_VEL
LIN {X 0,Y 418.243,Z 419.387,A -85,B 0,C 180,E1 -10217.767,E2 -10217.767} C_VEL
LIN {X 0,Y 418.261,Z 419.386,A -85,B 0,C 180,E1 -10220.618,E2 -10220.618} C_VEL
LIN {X 0,Y 418.247,Z 419.389,A -85,B 0,C 180,E1 -10223.976,E2 -10223.976} C_VEL
LIN {X 0,Y 418.258,Z 419.383,A -85,B 0,C 180,E1 -10227.156,E2 -10227.156} C_VEL
LIN {X 0,Y 418.269,Z 419.383,A -85,B 0,C 180,E1 -10230.895,E2 -10230.895} C_VEL
LIN {X 0,Y 418.272,Z 419.386,A -85,B 0,C 180,E1 -10234.096,E2 -10234.096} C_VEL
LIN {X 0,Y 418.239,Z 419.386,A -85,B 0,C 180,E1 -10237.264,E2 -10237.264} C_VEL
LIN {X 0,Y 418.285,Z 419.384,A -85,B 0,C 180,E1 -10240.364,E2 -10240.364} C_VEL
LIN {X 0,Y 418.318,Z 419.376,A -85,B 0,C 180,E1 -10243.405,E2 -10243.405} C_VEL
LIN {X 0,Y 418.356,Z 419.371,A -85,B 0,C 180,E1 -10246.994,E2 -10246.994} C_VEL
LIN {X 0,Y 418.359,Z 419.374,A -85,B 0,C 180,E1 -10250.329,E2 -10250.329} C_VEL
LIN {X 0,Y 418.481,Z 419.355,A -85,B 0,C 180,E1 -10253.249,E2 -10253.249} C_VEL
LIN {X 0,Y 418.344,Z 419.373,A -85,B 0,C 180,E1 -10255.182,E2 -10255.182} C_VEL
LIN {X 0,Y 418.547,Z 419.352,A -85,B 0,C 180,E1 -10258.076,E2 -10258.076} C_VEL
LIN {X 0,Y 418.675,Z 419.336,A -85,B 0,C 180,E1 -10260,E2 -10260} C_VEL
LIN {X 0,Y 418.502,Z 419.353,A -85,B 0,C 180,E1 -10262.888,E2 -10262.888} C_VEL
LIN {X 0,Y 418.495,Z 419.354,A -85,B 0,C 180,E1 -10266.751,E2 -10266.751} C_VEL
LIN {X 0,Y 418.343,Z 419.376,A -85,B 0,C 180,E1 -10269.672,E2 -10269.672} C_VEL
LIN {X 0,Y 418.348,Z 419.372,A -85,B 0,C 180,E1 -10273.001,E2 -10273.001} C_VEL
LIN {X 0,Y 418.315,Z 419.376,A -85,B 0,C 180,E1 -10276.736,E2 -10276.736} C_VEL
LIN {X 0,Y 418.273,Z 419.386,A -85,B 0,C 180,E1 -10279.791,E2 -10279.791} C_VEL
LIN {X 0,Y 418.24,Z 419.386,A -85,B 0,C 180,E1 -10282.736,E2 -10282.736} C_VEL
LIN {X 0,Y 418.273,Z 419.386,A -85,B 0,C 180,E1 -10285.904,E2 -10285.904} C_VEL
LIN {X 0,Y 418.267,Z 419.382,A -85,B 0,C 180,E1 -10289.162,E2 -10289.162} C_VEL
LIN {X 0,Y 418.259,Z 419.383,A -85,B 0,C 180,E1 -10292.844,E2 -10292.844} C_VEL
LIN {X 0,Y 418.251,Z 419.387,A -85,B 0,C 180,E1 -10296.239,E2 -10296.239} C_VEL
LIN {X 0,Y 418.255,Z 419.388,A -85,B 0,C 180,E1 -10299.682,E2 -10299.682} C_VEL
LIN {X 0,Y 418.234,Z 419.388,A -85,B 0,C 180,E1 -10302.322,E2 -10302.322} C_VEL
LIN {X 0,Y 418.245,Z 419.386,A -85,B 0,C 180,E1 -10305.11,E2 -10305.11} C_VEL
LIN {X 0,Y 418.245,Z 419.39,A -85,B 0,C 180,E1 -10307.767,E2 -10307.767} C_VEL
LIN {X 0,Y 418.26,Z 419.383,A -85,B 0,C 180,E1 -10310.619,E2 -10310.619} C_VEL
LIN {X 0,Y 418.249,Z 419.389,A -85,B 0,C 180,E1 -10313.977,E2 -10313.977} C_VEL
LIN {X 0,Y 418.263,Z 419.384,A -85,B 0,C 180,E1 -10317.156,E2 -10317.156} C_VEL
LIN {X 0,Y 418.278,Z 419.381,A -85,B 0,C 180,E1 -10320.839,E2 -10320.839} C_VEL
LIN {X 0,Y 418.274,Z 419.384,A -85,B 0,C 180,E1 -10324.096,E2 -10324.096} C_VEL
LIN {X 0,Y 418.242,Z 419.387,A -85,B 0,C 180,E1 -10327.264,E2 -10327.264} C_VEL
LIN {X 0,Y 418.287,Z 419.381,A -85,B 0,C 180,E1 -10330.365,E2 -10330.365} C_VEL
LIN {X 0,Y 418.321,Z 419.379,A -85,B 0,C 180,E1 -10333.405,E2 -10333.405} C_VEL
LIN {X 0,Y 418.355,Z 419.486,A -85,B 0,C 180,E1 -10336.781,E2 -10336.781} C_VEL
LIN {X 0,Y 421.734,Z 430.889,A -85,B 0,C 180,E1 -10337.611,E2 -10337.611} C_VEL
LIN {X 0,Y 422.441,Z 434.172,A -85,B 0,C 180,E1 -10337.876,E2 -10337.876} C_VEL
LIN {X 0,Y 421.868,Z 445.895,A -85,B 0,C 180,E1 -10338.833,E2 -10338.833} C_VEL
LIN {X 0,Y 421.255,Z 456.39,A -85,B 0,C 180,E1 -10339.921,E2 -10339.921} C_VEL
LIN {X 0,Y 420.574,Z 465.758,A -85,B 0,C 180,E1 -10341.116,E2 -10341.116} C_VEL
LIN {X 0,Y 420.016,Z 473.38,A -85,B 0,C 180,E1 -10342.307,E2 -10342.307} C_VEL
LIN {X 0,Y 419.517,Z 480.866,A -85,B 0,C 180,E1 -10343.749,E2 -10343.749} C_VEL
LIN {X 0,Y 419.046,Z 486.879,A -85,B 0,C 180,E1 -10345.19,E2 -10345.19} C_VEL
LIN {X 0,Y 418.671,Z 491.655,A -85,B 0,C 180,E1 -10346.632,E2 -10346.632} C_VEL
LIN {X 0,Y 418.406,Z 495.34,A -85,B 0,C 180,E1 -10348.075,E2 -10348.075} C_VEL
LIN {X 0,Y 418.175,Z 498.742,A -85,B 0,C 180,E1 -10350,E2 -10350} C_VEL
LIN {X 0,Y 418.029,Z 499.825,A -85,B 0,C 180,E1 -10350.964,E2 -10350.964} C_VEL
LIN {X 0,Y 418.075,Z 500.49,A -85,B 0,C 180,E1 -10351.927,E2 -10351.927} C_VEL
LIN {X 0,Y 418.017,Z 500.746,A -85,B 0,C 180,E1 -10353.856,E2 -10353.856} C_VEL
LIN {X 0,Y 418.107,Z 500.269,A -85,B 0,C 180,E1 -10354.821,E2 -10354.821} C_VEL
LIN {X 0,Y 418.301,Z 499.384,A -85,B 0,C 180,E1 -10355.786,E2 -10355.786} C_VEL
LIN {X 0,Y 418.459,Z 497.119,A -85,B 0,C 180,E1 -10357.353,E2 -10357.353} C_VEL
LIN {X 0,Y 417.958,Z 495.763,A -85,B 0,C 180,E1 -10358.139,E2 -10358.139} C_VEL
LIN {X 0,Y 415.409,Z 493.267,A -85,B 0,C 180,E1 -10359.413,E2 -10359.413} C_VEL
LIN {X 0,Y 412.921,Z 490.04,A -85,B 0,C 180,E1 -10360.666,E2 -10360.666} C_VEL
LIN {X 0,Y 412.517,Z 487.523,A -85,B 0,C 180,E1 -10361.407,E2 -10361.407} C_VEL
LIN {X 0,Y 413.007,Z 480.724,A -85,B 0,C 180,E1 -10363.031,E2 -10363.031} C_VEL
LIN {X 0,Y 413.693,Z 473.153,A -85,B 0,C 180,E1 -10364.454,E2 -10364.454} C_VEL
LIN {X 0,Y 414.386,Z 464.714,A -85,B 0,C 180,E1 -10365.746,E2 -10365.746} C_VEL
LIN {X 0,Y 415.064,Z 454.768,A -85,B 0,C 180,E1 -10366.983,E2 -10366.983} C_VEL
LIN {X 0,Y 415.836,Z 443.445,A -85,B 0,C 180,E1 -10368.091,E2 -10368.091} C_VEL
LIN {X 0,Y 416.019,Z 435.774,A -85,B 0,C 180,E1 -10368.722,E2 -10368.722} C_VEL
LIN {X 0,Y 413.026,Z 425.704,A -85,B 0,C 180,E1 -10369.565,E2 -10369.565} C_VEL
LIN {X 0,Y 411.223,Z 420.263,A -85,B 0,C 180,E1 -10369.987,E2 -10369.987} C_VEL
LIN {X 0,Y 411.2,Z 420.26,A -85,B 0,C 180,E1 -10373.148,E2 -10373.148} C_VEL
LIN {X 0,Y 411.241,Z 420.261,A -85,B 0,C 180,E1 -10376.381,E2 -10376.381} C_VEL
LIN {X 0,Y 411.205,Z 420.261,A -85,B 0,C 180,E1 -10379.713,E2 -10379.713} C_VEL
LIN {X 0,Y 411.211,Z 420.259,A -85,B 0,C 180,E1 -10383.156,E2 -10383.156} C_VEL
LIN {X 0,Y 411.198,Z 420.263,A -85,B 0,C 180,E1 -10386.553,E2 -10386.553} C_VEL
LIN {X 0,Y 411.217,Z 420.26,A -85,B 0,C 180,E1 -10389.728,E2 -10389.728} C_VEL
LIN {X 0,Y 411.178,Z 420.263,A -85,B 0,C 180,E1 -10393.134,E2 -10393.134} C_VEL
LIN {X 0,Y 411.174,Z 420.268,A -85,B 0,C 180,E1 -10395.881,E2 -10395.881} C_VEL
LIN {X 0,Y 411.168,Z 420.264,A -85,B 0,C 180,E1 -10398.772,E2 -10398.772} C_VEL
LIN {X 0,Y 411.199,Z 420.267,A -85,B 0,C 180,E1 -10402.026,E2 -10402.026} C_VEL
LIN {X 0,Y 411.21,Z 420.263,A -85,B 0,C 180,E1 -10405.667,E2 -10405.667} C_VEL
LIN {X 0,Y 411.194,Z 420.261,A -85,B 0,C 180,E1 -10409.152,E2 -10409.152} C_VEL
LIN {X 0,Y 411.263,Z 420.253,A -85,B 0,C 180,E1 -10412.522,E2 -10412.522} C_VEL
LIN {X 0,Y 411.224,Z 420.264,A -85,B 0,C 180,E1 -10415.784,E2 -10415.784} C_VEL
LIN {X 0,Y 411.201,Z 420.26,A -85,B 0,C 180,E1 -10418.966,E2 -10418.966} C_VEL
LIN {X 0,Y 411.255,Z 420.256,A -85,B 0,C 180,E1 -10422.085,E2 -10422.085} C_VEL
LIN {X 0,Y 411.305,Z 420.274,A -85,B 0,C 180,E1 -10425.07,E2 -10425.07} C_VEL
LIN {X 0,Y 414.52,Z 432.655,A -85,B 0,C 180,E1 -10425.997,E2 -10425.997} C_VEL
LIN {X 0,Y 414.104,Z 444.767,A -85,B 0,C 180,E1 -10427.004,E2 -10427.004} C_VEL
LIN {X 0,Y 413.479,Z 455.404,A -85,B 0,C 180,E1 -10428.106,E2 -10428.106} C_VEL
LIN {X 0,Y 413.069,Z 464.161,A -85,B 0,C 180,E1 -10429.213,E2 -10429.213} C_VEL
LIN {X 0,Y 412.47,Z 473.771,A -85,B 0,C 180,E1 -10430.684,E2 -10430.684} C_VEL
LIN {X 0,Y 412.053,Z 481.448,A -85,B 0,C 180,E1 -10432.157,E2 -10432.157} C_VEL
LIN {X 0,Y 411.645,Z 487.66,A -85,B 0,C 180,E1 -10433.628,E2 -10433.628} C_VEL
LIN {X 0,Y 411.27,Z 492.621,A -85,B 0,C 180,E1 -10435.098,E2 -10435.098} C_VEL
LIN {X 0,Y 411.159,Z 496.438,A -85,B 0,C 180,E1 -10436.57,E2 -10436.57} C_VEL
LIN {X 0,Y 411.071,Z 499.237,A -85,B 0,C 180,E1 -10438.04,E2 -10438.04} C_VEL
LIN {X 0,Y 410.981,Z 500.601,A -85,B 0,C 180,E1 -10439.02,E2 -10439.02} C_VEL
LIN {X 0,Y 411.045,Z 501.489,A -85,B 0,C 180,E1 -10440,E2 -10440} C_VEL
LIN {X 0,Y 411.174,Z 502.123,A -85,B 0,C 180,E1 -10441.959,E2 -10441.959} C_VEL
LIN {X 0,Y 411.181,Z 501.819,A -85,B 0,C 180,E1 -10442.939,E2 -10442.939} C_VEL
LIN {X 0,Y 411.37,Z 500.004,A -85,B 0,C 180,E1 -10444.9,E2 -10444.9} C_VEL
LIN {X 0,Y 411.79,Z 497.493,A -85,B 0,C 180,E1 -10446.369,E2 -10446.369} C_VEL
LIN {X 0,Y 412.176,Z 493.985,A -85,B 0,C 180,E1 -10447.84,E2 -10447.84} C_VEL
LIN {X 0,Y 412.602,Z 489.38,A -85,B 0,C 180,E1 -10449.312,E2 -10449.312} C_VEL
LIN {X 0,Y 413.228,Z 482.358,A -85,B 0,C 180,E1 -10451.031,E2 -10451.031} C_VEL
LIN {X 0,Y 413.964,Z 474.713,A -85,B 0,C 180,E1 -10452.501,E2 -10452.501} C_VEL
LIN {X 0,Y 414.769,Z 465.06,A -85,B 0,C 180,E1 -10453.972,E2 -10453.972} C_VEL
LIN {X 0,Y 415.511,Z 455.517,A -85,B 0,C 180,E1 -10455.144,E2 -10455.144} C_VEL
LIN {X 0,Y 416.396,Z 443.779,A -85,B 0,C 180,E1 -10456.296,E2 -10456.296} C_VEL
LIN {X 0,Y 416.777,Z 436.584,A -85,B 0,C 180,E1 -10456.881,E2 -10456.881} C_VEL
LIN {X 0,Y 413.437,Z 426.233,A -85,B 0,C 180,E1 -10457.834,E2 -10457.834} C_VEL
LIN {X 0,Y 411.265,Z 420.264,A -85,B 0,C 180,E1 -10458.365,E2 -10458.365} C_VEL
LIN {X 0,Y 411.2,Z 420.27,A -85,B 0,C 180,E1 -10461.034,E2 -10461.034} C_VEL
LIN {X 0,Y 411.229,Z 420.261,A -85,B 0,C 180,E1 -10464.215,E2 -10464.215} C_VEL
LIN {X 0,Y 411.262,Z 420.256,A -85,B 0,C 180,E1 -10467.477,E2 -10467.477} C_VEL
LIN {X 0,Y 411.193,Z 420.267,A -85,B 0,C 180,E1 -10470.847,E2 -10470.847} C_VEL
LIN {X 0,Y 411.209,Z 420.266,A -85,B 0,C 180,E1 -10474.333,E2 -10474.333} C_VEL
LIN {X 0,Y 411.197,Z 420.265,A -85,B 0,C 180,E1 -10477.973,E2 -10477.973} C_VEL
LIN {X 0,Y 411.167,Z 420.266,A -85,B 0,C 180,E1 -10481.228,E2 -10481.228} C_VEL
LIN {X 0,Y 411.179,Z 420.267,A -85,B 0,C 180,E1 -10484.49,E2 -10484.49} C_VEL
LIN {X 0,Y 411.191,Z 420.276,A -85,B 0,C 180,E1 -10486.79,E2 -10486.79} C_VEL
LIN {X 0,Y 413.063,Z 429.345,A -85,B 0,C 180,E1 -10489.965,E2 -10489.965} C_VEL
LIN {X 0,Y 414.652,Z 438.029,A -85,B 0,C 180,E1 -10492.808,E2 -10492.808} C_VEL
LIN {X 0,Y 414.193,Z 444.644,A -85,B 0,C 180,E1 -10494.766,E2 -10494.766} C_VEL
LIN {X 0,Y 413.306,Z 456.721,A -85,B 0,C 180,E1 -10498.235,E2 -10498.235} C_VEL
LIN {X 0,Y 412.407,Z 470.313,A -85,B 0,C 180,E1 -10502.013,E2 -10502.013} C_VEL
LIN {X 0,Y 411.672,Z 484.275,A -85,B 0,C 180,E1 -10505.812,E2 -10505.812} C_VEL
LIN {X 0,Y 411.132,Z 495.988,A -85,B 0,C 180,E1 -10508.962,E2 -10508.962} C_VEL
LIN {X 0,Y 410.77,Z 508.041,A -85,B 0,C 180,E1 -10512.213,E2 -10512.213} C_VEL
LIN {X 0,Y 412.561,Z 522.656,A -85,B 0,C 180,E1 -10512.7,E2 -10512.7} C_VEL
LIN {X 0,Y 413.451,Z 534.82,A -85,B 0,C 180,E1 -10513.267,E2 -10513.267} C_VEL
LIN {X 0,Y 414.023,Z 546.602,A -85,B 0,C 180,E1 -10513.988,E2 -10513.988} C_VEL
LIN {X 0,Y 413.292,Z 558.048,A -85,B 0,C 180,E1 -10514.844,E2 -10514.844} C_VEL
LIN {X 0,Y 412.405,Z 569.715,A -85,B 0,C 180,E1 -10515.945,E2 -10515.945} C_VEL
LIN {X 0,Y 411.83,Z 578.993,A -85,B 0,C 180,E1 -10517.033,E2 -10517.033} C_VEL
LIN {X 0,Y 411.16,Z 588.585,A -85,B 0,C 180,E1 -10518.413,E2 -10518.413} C_VEL
LIN {X 0,Y 410.667,Z 596.93,A -85,B 0,C 180,E1 -10519.897,E2 -10519.897} C_VEL
LIN {X 0,Y 410.474,Z 603.697,A -85,B 0,C 180,E1 -10521.384,E2 -10521.384} C_VEL
LIN {X 0,Y 410.434,Z 609.893,A -85,B 0,C 180,E1 -10523.116,E2 -10523.116} C_VEL
LIN {X 0,Y 410.485,Z 613.946,A -85,B 0,C 180,E1 -10524.596,E2 -10524.596} C_VEL
LIN {X 0,Y 410.642,Z 616.955,A -85,B 0,C 180,E1 -10526.074,E2 -10526.074} C_VEL
LIN {X 0,Y 410.638,Z 619.382,A -85,B 0,C 180,E1 -10528.038,E2 -10528.038} C_VEL
LIN {X 0,Y 410.872,Z 620.024,A -85,B 0,C 180,E1 -10529.02,E2 -10529.02} C_VEL
LIN {X 0,Y 410.882,Z 620.204,A -85,B 0,C 180,E1 -10530,E2 -10530} C_VEL
LIN {X 0,Y 410.874,Z 619.951,A -85,B 0,C 180,E1 -10530.98,E2 -10530.98} C_VEL
LIN {X 0,Y 410.628,Z 618.207,A -85,B 0,C 180,E1 -10532.943,E2 -10532.943} C_VEL
LIN {X 0,Y 410.64,Z 616.707,A -85,B 0,C 180,E1 -10533.925,E2 -10533.925} C_VEL
LIN {X 0,Y 410.527,Z 613.596,A -85,B 0,C 180,E1 -10535.403,E2 -10535.403} C_VEL
LIN {X 0,Y 410.46,Z 609.399,A -85,B 0,C 180,E1 -10536.884,E2 -10536.884} C_VEL
LIN {X 0,Y 410.516,Z 602.967,A -85,B 0,C 180,E1 -10538.615,E2 -10538.615} C_VEL
LIN {X 0,Y 410.708,Z 595.985,A -85,B 0,C 180,E1 -10540.102,E2 -10540.102} C_VEL
LIN {X 0,Y 411.149,Z 587.344,A -85,B 0,C 180,E1 -10541.586,E2 -10541.586} C_VEL
LIN {X 0,Y 411.783,Z 578.485,A -85,B 0,C 180,E1 -10542.819,E2 -10542.819} C_VEL
LIN {X 0,Y 412.099,Z 571.444,A -85,B 0,C 180,E1 -10543.651,E2 -10543.651} C_VEL
LIN {X 0,Y 412.829,Z 561.121,A -85,B 0,C 180,E1 -10544.669,E2 -10544.669} C_VEL
LIN {X 0,Y 413.596,Z 550.281,A -85,B 0,C 180,E1 -10545.523,E2 -10545.523} C_VEL
LIN {X 0,Y 413.807,Z 546.698,A -85,B 0,C 180,E1 -10545.768,E2 -10545.768} C_VEL
LIN {X 0,Y 413.031,Z 535.029,A -85,B 0,C 180,E1 -10546.473,E2 -10546.473} C_VEL
LIN {X 0,Y 412.097,Z 521.695,A -85,B 0,C 180,E1 -10547.068,E2 -10547.068} C_VEL
LIN {X 0,Y 410.747,Z 508.405,A -85,B 0,C 180,E1 -10547.478,E2 -10547.478} C_VEL
LIN {X 0,Y 411.122,Z 495.008,A -85,B 0,C 180,E1 -10551.038,E2 -10551.038} C_VEL
LIN {X 0,Y 411.698,Z 481.22,A -85,B 0,C 180,E1 -10554.713,E2 -10554.713} C_VEL
LIN {X 0,Y 412.259,Z 469.069,A -85,B 0,C 180,E1 -10557.975,E2 -10557.975} C_VEL
LIN {X 0,Y 412.868,Z 459.036,A -85,B 0,C 180,E1 -10560.708,E2 -10560.708} C_VEL
LIN {X 0,Y 413.704,Z 445.837,A -85,B 0,C 180,E1 -10564.392,E2 -10564.392} C_VEL
LIN {X 0,Y 414.321,Z 437.571,A -85,B 0,C 180,E1 -10566.768,E2 -10566.768} C_VEL
LIN {X 0,Y 413.483,Z 431.785,A -85,B 0,C 180,E1 -10568.568,E2 -10568.568} C_VEL
LIN {X 0,Y 411.86,Z 423.324,A -85,B 0,C 180,E1 -10571.339,E2 -10571.339} C_VEL
LIN {X 0,Y 411.195,Z 420.266,A -85,B 0,C 180,E1 -10572.436,E2 -10572.436} C_VEL
LIN {X 0,Y 411.173,Z 420.27,A -85,B 0,C 180,E1 -10575.88,E2 -10575.88} C_VEL
LIN {X 0,Y 411.167,Z 420.268,A -85,B 0,C 180,E1 -10578.771,E2 -10578.771} C_VEL
LIN {X 0,Y 411.212,Z 420.264,A -85,B 0,C 180,E1 -10581.83,E2 -10581.83} C_VEL
LIN {X 0,Y 411.212,Z 420.261,A -85,B 0,C 180,E1 -10585.121,E2 -10585.121} C_VEL
LIN {X 0,Y 411.166,Z 420.271,A -85,B 0,C 180,E1 -10588.003,E2 -10588.003} C_VEL
LIN {X 0,Y 411.219,Z 420.26,A -85,B 0,C 180,E1 -10591.41,E2 -10591.41} C_VEL
LIN {X 0,Y 411.239,Z 420.259,A -85,B 0,C 180,E1 -10593.619,E2 -10593.619} C_VEL
LIN {X 0,Y 411.204,Z 420.262,A -85,B 0,C 180,E1 -10596.853,E2 -10596.853} C_VEL
LIN {X 0,Y 411.216,Z 420.265,A -85,B 0,C 180,E1 -10600.05,E2 -10600.05} C_VEL
LIN {X 0,Y 411.264,Z 420.254,A -85,B 0,C 180,E1 -10603.131,E2 -10603.131} C_VEL
LIN {X 0,Y 411.315,Z 420.249,A -85,B 0,C 180,E1 -10606.891,E2 -10606.891} C_VEL
LIN {X 0,Y 411.308,Z 420.254,A -85,B 0,C 180,E1 -10610.162,E2 -10610.162} C_VEL
LIN {X 0,Y 411.444,Z 420.232,A -85,B 0,C 180,E1 -10613.133,E2 -10613.133} C_VEL
LIN {X 0,Y 411.314,Z 420.248,A -85,B 0,C 180,E1 -10615.099,E2 -10615.099} C_VEL
LIN {X 0,Y 411.516,Z 420.228,A -85,B 0,C 180,E1 -10618.043,E2 -10618.043} C_VEL
LIN {X 0,Y 411.644,Z 420.212,A -85,B 0,C 180,E1 -10620,E2 -10620} C_VEL
LIN {X 0,Y 411.459,Z 420.23,A -85,B 0,C 180,E1 -10622.937,E2 -10622.937} C_VEL
LIN {X 0,Y 411.462,Z 420.23,A -85,B 0,C 180,E1 -10626.867,E2 -10626.867} C_VEL
LIN {X 0,Y 411.295,Z 420.255,A -85,B 0,C 180,E1 -10629.839,E2 -10629.839} C_VEL
LIN {X 0,Y 411.307,Z 420.249,A -85,B 0,C 180,E1 -10633.104,E2 -10633.104} C_VEL
LIN {X 0,Y 411.264,Z 420.254,A -85,B 0,C 180,E1 -10636.869,E2 -10636.869} C_VEL
LIN {X 0,Y 411.232,Z 420.263,A -85,B 0,C 180,E1 -10639.987,E2 -10639.987} C_VEL
LIN {X 0,Y 411.205,Z 420.262,A -85,B 0,C 180,E1 -10643.148,E2 -10643.148} C_VEL
LIN {X 0,Y 411.24,Z 420.259,A -85,B 0,C 180,E1 -10646.381,E2 -10646.381} C_VEL
LIN {X 0,Y 411.202,Z 420.267,A -85,B 0,C 180,E1 -10649.713,E2 -10649.713} C_VEL
LIN {X 0,Y 411.208,Z 420.262,A -85,B 0,C 180,E1 -10653.156,E2 -10653.156} C_VEL
LIN {X 0,Y 411.197,Z 420.263,A -85,B 0,C 180,E1 -10656.553,E2 -10656.553} C_VEL
LIN {X 0,Y 411.218,Z 420.264,A -85,B 0,C 180,E1 -10659.729,E2 -10659.729} C_VEL
LIN {X 0,Y 411.18,Z 420.265,A -85,B 0,C 180,E1 -10663.133,E2 -10663.133} C_VEL
LIN {X 0,Y 411.176,Z 420.27,A -85,B 0,C 180,E1 -10665.88,E2 -10665.88} C_VEL
LIN {X 0,Y 411.167,Z 420.266,A -85,B 0,C 180,E1 -10668.772,E2 -10668.772} C_VEL
LIN {X 0,Y 411.213,Z 420.265,A -85,B 0,C 180,E1 -10671.831,E2 -10671.831} C_VEL
LIN {X 0,Y 411.214,Z 420.261,A -85,B 0,C 180,E1 -10675.122,E2 -10675.122} C_VEL
LIN {X 0,Y 411.175,Z 420.269,A -85,B 0,C 180,E1 -10678.004,E2 -10678.004} C_VEL
LIN {X 0,Y 411.228,Z 420.262,A -85,B 0,C 180,E1 -10681.411,E2 -10681.411} C_VEL
LIN {X 0,Y 411.24,Z 420.257,A -85,B 0,C 180,E1 -10684.707,E2 -10684.707} C_VEL
LIN {X 0,Y 411.209,Z 420.265,A -85,B 0,C 180,E1 -10687.914,E2 -10687.914} C_VEL
LIN {X 0,Y 411.229,Z 420.26,A -85,B 0,C 180,E1 -10691.052,E2 -10691.052} C_VEL
LIN {X 0,Y 411.259,Z 420.257,A -85,B 0,C 180,E1 -10694.132,E2 -10694.132} C_VEL
LIN {X 0,Y 411.316,Z 420.391,A -85,B 0,C 180,E1 -10696.508,E2 -10696.508} C_VEL
LIN {X 0,Y 414.406,Z 430.702,A -85,B 0,C 180,E1 -10697.264,E2 -10697.264} C_VEL
LIN {X 0,Y 415.618,Z 435.654,A -85,B 0,C 180,E1 -10697.673,E2 -10697.673} C_VEL
LIN {X 0,Y 415.019,Z 447.248,A -85,B 0,C 180,E1 -10698.647,E2 -10698.647} C_VEL
LIN {X 0,Y 414.394,Z 457.45,A -85,B 0,C 180,E1 -10699.724,E2 -10699.724} C_VEL
LIN {X 0,Y 413.668,Z 466.947,A -85,B 0,C 180,E1 -10700.959,E2 -10700.959} C_VEL
LIN {X 0,Y 413.064,Z 475.903,A -85,B 0,C 180,E1 -10702.423,E2 -10702.423} C_VEL
LIN {X 0,Y 412.422,Z 483.119,A -85,B 0,C 180,E1 -10703.886,E2 -10703.886} C_VEL
LIN {X 0,Y 411.954,Z 489.74,A -85,B 0,C 180,E1 -10705.597,E2 -10705.597} C_VEL
LIN {X 0,Y 411.598,Z 494.113,A -85,B 0,C 180,E1 -10707.064,E2 -10707.064} C_VEL
LIN {X 0,Y 411.394,Z 496.422,A -85,B 0,C 180,E1 -10708.042,E2 -10708.042} C_VEL
LIN {X 0,Y 411.156,Z 499.799,A -85,B 0,C 180,E1 -10710,E2 -10710} C_VEL
LIN {X 0,Y 411.03,Z 500.859,A -85,B 0,C 180,E1 -10710.98,E2 -10710.98} C_VEL
LIN {X 0,Y 411.052,Z 501.517,A -85,B 0,C 180,E1 -10711.96,E2 -10711.96} C_VEL
LIN {X 0,Y 410.996,Z 501.752,A -85,B 0,C 180,E1 -10713.922,E2 -10713.922} C_VEL
LIN {X 0,Y 411.303,Z 500.358,A -85,B 0,C 180,E1 -10715.885,E2 -10715.885} C_VEL
LIN {X 0,Y 411.53,Z 497.446,A -85,B 0,C 180,E1 -10717.853,E2 -10717.853} C_VEL
LIN {X 0,Y 411.851,Z 494.106,A -85,B 0,C 180,E1 -10719.33,E2 -10719.33} C_VEL
LIN {X 0,Y 412.335,Z 489.684,A -85,B 0,C 180,E1 -10720.807,E2 -10720.807} C_VEL
LIN {X 0,Y 412.517,Z 487.523,A -85,B 0,C 180,E1 -10721.407,E2 -10721.407} C_VEL
LIN {X 0,Y 412.13,Z 484.852,A -85,B 0,C 180,E1 -10722.134,E2 -10722.134} C_VEL
LIN {X 0,Y 409.761,Z 480.298,A -85,B 0,C 180,E1 -10723.321,E2 -10723.321} C_VEL
LIN {X 0,Y 407.435,Z 475.183,A -85,B 0,C 180,E1 -10724.464,E2 -10724.464} C_VEL
LIN {X 0,Y 407.104,Z 471.514,A -85,B 0,C 180,E1 -10725.111,E2 -10725.111} C_VEL
LIN {X 0,Y 407.884,Z 461.733,A -85,B 0,C 180,E1 -10726.517,E2 -10726.517} C_VEL
LIN {X 0,Y 408.565,Z 451.987,A -85,B 0,C 180,E1 -10727.649,E2 -10727.649} C_VEL
LIN {X 0,Y 409.283,Z 440.421,A -85,B 0,C 180,E1 -10728.71,E2 -10728.71} C_VEL
LIN {X 0,Y 409.338,Z 437.634,A -85,B 0,C 180,E1 -10728.939,E2 -10728.939} C_VEL
LIN {X 0,Y 406.404,Z 427.887,A -85,B 0,C 180,E1 -10729.791,E2 -10729.791} C_VEL
LIN {X 0,Y 404.161,Z 421.144,A -85,B 0,C 180,E1 -10730.321,E2 -10730.321} C_VEL
LIN {X 0,Y 404.168,Z 421.136,A -85,B 0,C 180,E1 -10733.575,E2 -10733.575} C_VEL
LIN {X 0,Y 404.187,Z 421.135,A -85,B 0,C 180,E1 -10735.767,E2 -10735.767} C_VEL
LIN {X 0,Y 404.2,Z 421.136,A -85,B 0,C 180,E1 -10738,E2 -10738} C_VEL
LIN {X 0,Y 404.144,Z 421.14,A -85,B 0,C 180,E1 -10741.558,E2 -10741.558} C_VEL
LIN {X 0,Y 404.19,Z 421.134,A -85,B 0,C 180,E1 -10745.016,E2 -10745.016} C_VEL
LIN {X 0,Y 404.159,Z 421.138,A -85,B 0,C 180,E1 -10748.757,E2 -10748.757} C_VEL
LIN {X 0,Y 404.127,Z 421.143,A -85,B 0,C 180,E1 -10751.6,E2 -10751.6} C_VEL
LIN {X 0,Y 404.15,Z 421.141,A -85,B 0,C 180,E1 -10754.522,E2 -10754.522} C_VEL
LIN {X 0,Y 404.141,Z 421.14,A -85,B 0,C 180,E1 -10757.296,E2 -10757.296} C_VEL
LIN {X 0,Y 404.173,Z 421.142,A -85,B 0,C 180,E1 -10759.955,E2 -10759.955} C_VEL
LIN {X 0,Y 404.14,Z 421.14,A -85,B 0,C 180,E1 -10763.125,E2 -10763.125} C_VEL
LIN {X 0,Y 404.149,Z 421.142,A -85,B 0,C 180,E1 -10766.188,E2 -10766.188} C_VEL
LIN {X 0,Y 404.15,Z 421.143,A -85,B 0,C 180,E1 -10769.715,E2 -10769.715} C_VEL
LIN {X 0,Y 404.199,Z 421.133,A -85,B 0,C 180,E1 -10773.123,E2 -10773.123} C_VEL
LIN {X 0,Y 404.178,Z 421.137,A -85,B 0,C 180,E1 -10775.334,E2 -10775.334} C_VEL
LIN {X 0,Y 404.143,Z 421.139,A -85,B 0,C 180,E1 -10778.581,E2 -10778.581} C_VEL
LIN {X 0,Y 404.213,Z 421.138,A -85,B 0,C 180,E1 -10781.762,E2 -10781.762} C_VEL
LIN {X 0,Y 404.247,Z 421.126,A -85,B 0,C 180,E1 -10784.851,E2 -10784.851} C_VEL
LIN {X 0,Y 407.648,Z 434.62,A -85,B 0,C 180,E1 -10785.903,E2 -10785.903} C_VEL
LIN {X 0,Y 407.11,Z 446.337,A -85,B 0,C 180,E1 -10786.904,E2 -10786.904} C_VEL
LIN {X 0,Y 406.507,Z 456.839,A -85,B 0,C 180,E1 -10788.026,E2 -10788.026} C_VEL
LIN {X 0,Y 406.003,Z 466.418,A -85,B 0,C 180,E1 -10789.275,E2 -10789.275} C_VEL
LIN {X 0,Y 405.509,Z 474.356,A -85,B 0,C 180,E1 -10790.523,E2 -10790.523} C_VEL
LIN {X 0,Y 405.053,Z 482.142,A -85,B 0,C 180,E1 -10792.021,E2 -10792.021} C_VEL
LIN {X 0,Y 404.656,Z 488.423,A -85,B 0,C 180,E1 -10793.518,E2 -10793.518} C_VEL
LIN {X 0,Y 404.26,Z 493.456,A -85,B 0,C 180,E1 -10795.013,E2 -10795.013} C_VEL
LIN {X 0,Y 404.14,Z 497.336,A -85,B 0,C 180,E1 -10796.51,E2 -10796.51} C_VEL
LIN {X 0,Y 404.049,Z 500.192,A -85,B 0,C 180,E1 -10798.006,E2 -10798.006} C_VEL
LIN {X 0,Y 403.958,Z 501.592,A -85,B 0,C 180,E1 -10799.003,E2 -10799.003} C_VEL
LIN {X 0,Y 404.036,Z 502.513,A -85,B 0,C 180,E1 -10800,E2 -10800} C_VEL
LIN {X 0,Y 404.173,Z 503.2,A -85,B 0,C 180,E1 -10801.993,E2 -10801.993} C_VEL
LIN {X 0,Y 404.179,Z 502.934,A -85,B 0,C 180,E1 -10802.99,E2 -10802.99} C_VEL
LIN {X 0,Y 404.392,Z 501.178,A -85,B 0,C 180,E1 -10804.985,E2 -10804.985} C_VEL
LIN {X 0,Y 404.62,Z 499.674,A -85,B 0,C 180,E1 -10805.982,E2 -10805.982} C_VEL
LIN {X 0,Y 405.113,Z 496.551,A -85,B 0,C 180,E1 -10807.476,E2 -10807.476} C_VEL
LIN {X 0,Y 405.533,Z 492.369,A -85,B 0,C 180,E1 -10808.973,E2 -10808.973} C_VEL
LIN {X 0,Y 406.201,Z 485.95,A -85,B 0,C 180,E1 -10810.719,E2 -10810.719} C_VEL
LIN {X 0,Y 406.956,Z 478.884,A -85,B 0,C 180,E1 -10812.213,E2 -10812.213} C_VEL
LIN {X 0,Y 407.787,Z 470.095,A -85,B 0,C 180,E1 -10813.708,E2 -10813.708} C_VEL
LIN {X 0,Y 408.545,Z 461.069,A -85,B 0,C 180,E1 -10814.954,E2 -10814.954} C_VEL
LIN {X 0,Y 409.514,Z 449.992,A -85,B 0,C 180,E1 -10816.167,E2 -10816.167} C_VEL
LIN {X 0,Y 410.242,Z 438.619,A -85,B 0,C 180,E1 -10817.167,E2 -10817.167} C_VEL
LIN {X 0,Y 406.836,Z 428.273,A -85,B 0,C 180,E1 -10818.173,E2 -10818.173} C_VEL
LIN {X 0,Y 404.185,Z 421.146,A -85,B 0,C 180,E1 -10818.83,E2 -10818.83} C_VEL
LIN {X 0,Y 404.142,Z 421.149,A -85,B 0,C 180,E1 -10821.419,E2 -10821.419} C_VEL
LIN {X 0,Y 404.18,Z 421.14,A -85,B 0,C 180,E1 -10824.665,E2 -10824.665} C_VEL
LIN {X 0,Y 404.199,Z 421.135,A -85,B 0,C 180,E1 -10827.999,E2 -10827.999} C_VEL
LIN {X 0,Y 404.142,Z 421.143,A -85,B 0,C 180,E1 -10831.558,E2 -10831.558} C_VEL
LIN {X 0,Y 404.188,Z 421.139,A -85,B 0,C 180,E1 -10835.016,E2 -10835.016} C_VEL
LIN {X 0,Y 404.157,Z 421.142,A -85,B 0,C 180,E1 -10838.757,E2 -10838.757} C_VEL
LIN {X 0,Y 404.126,Z 421.141,A -85,B 0,C 180,E1 -10841.6,E2 -10841.6} C_VEL
LIN {X 0,Y 404.148,Z 421.142,A -85,B 0,C 180,E1 -10844.522,E2 -10844.522} C_VEL
LIN {X 0,Y 404.161,Z 421.273,A -85,B 0,C 180,E1 -10846.441,E2 -10846.441} C_VEL
LIN {X 0,Y 405.991,Z 430.059,A -85,B 0,C 180,E1 -10849.612,E2 -10849.612} C_VEL
LIN {X 0,Y 407.61,Z 438.635,A -85,B 0,C 180,E1 -10852.479,E2 -10852.479} C_VEL
LIN {X 0,Y 407.668,Z 441.927,A -85,B 0,C 180,E1 -10853.504,E2 -10853.504} C_VEL
LIN {X 0,Y 406.565,Z 453.779,A -85,B 0,C 180,E1 -10857.008,E2 -10857.008} C_VEL
LIN {X 0,Y 405.777,Z 464.188,A -85,B 0,C 180,E1 -10859.997,E2 -10859.997} C_VEL
LIN {X 0,Y 405.103,Z 475.537,A -85,B 0,C 180,E1 -10863.188,E2 -10863.188} C_VEL
LIN {X 0,Y 404.489,Z 487.301,A -85,B 0,C 180,E1 -10866.445,E2 -10866.445} C_VEL
LIN {X 0,Y 403.92,Z 500.123,A -85,B 0,C 180,E1 -10869.98,E2 -10869.98} C_VEL
LIN {X 0,Y 403.708,Z 506.98,A -85,B 0,C 180,E1 -10871.865,E2 -10871.865} C_VEL
LIN {X 0,Y 405.617,Z 522.178,A -85,B 0,C 180,E1 -10872.394,E2 -10872.394} C_VEL
LIN {X 0,Y 406.481,Z 534.162,A -85,B 0,C 180,E1 -10872.971,E2 -10872.971} C_VEL
LIN {X 0,Y 406.998,Z 545.825,A -85,B 0,C 180,E1 -10873.704,E2 -10873.704} C_VEL
LIN {X 0,Y 406.657,Z 554.271,A -85,B 0,C 180,E1 -10874.333,E2 -10874.333} C_VEL
LIN {X 0,Y 405.73,Z 565.291,A -85,B 0,C 180,E1 -10875.325,E2 -10875.325} C_VEL
LIN {X 0,Y 404.91,Z 575.654,A -85,B 0,C 180,E1 -10876.494,E2 -10876.494} C_VEL
LIN {X 0,Y 404.314,Z 584.451,A -85,B 0,C 180,E1 -10877.705,E2 -10877.705} C_VEL
LIN {X 0,Y 403.758,Z 593.43,A -85,B 0,C 180,E1 -10879.215,E2 -10879.215} C_VEL
LIN {X 0,Y 403.468,Z 600.656,A -85,B 0,C 180,E1 -10880.728,E2 -10880.728} C_VEL
LIN {X 0,Y 403.368,Z 607.312,A -85,B 0,C 180,E1 -10882.491,E2 -10882.491} C_VEL
LIN {X 0,Y 403.413,Z 611.728,A -85,B 0,C 180,E1 -10884,E2 -10884} C_VEL
LIN {X 0,Y 403.494,Z 614.083,A -85,B 0,C 180,E1 -10885.004,E2 -10885.004} C_VEL
LIN {X 0,Y 403.602,Z 615.964,A -85,B 0,C 180,E1 -10886.006,E2 -10886.006} C_VEL
LIN {X 0,Y 403.599,Z 618.382,A -85,B 0,C 180,E1 -10888.004,E2 -10888.004} C_VEL
LIN {X 0,Y 403.846,Z 619.02,A -85,B 0,C 180,E1 -10889.003,E2 -10889.003} C_VEL
LIN {X 0,Y 403.861,Z 619.19,A -85,B 0,C 180,E1 -10890,E2 -10890} C_VEL
LIN {X 0,Y 403.848,Z 618.93,A -85,B 0,C 180,E1 -10890.997,E2 -10890.997} C_VEL
LIN {X 0,Y 403.587,Z 617.172,A -85,B 0,C 180,E1 -10892.994,E2 -10892.994} C_VEL
LIN {X 0,Y 403.603,Z 615.66,A -85,B 0,C 180,E1 -10893.994,E2 -10893.994} C_VEL
LIN {X 0,Y 403.45,Z 612.529,A -85,B 0,C 180,E1 -10895.498,E2 -10895.498} C_VEL
LIN {X 0,Y 403.396,Z 608.318,A -85,B 0,C 180,E1 -10897.005,E2 -10897.005} C_VEL
LIN {X 0,Y 403.462,Z 601.867,A -85,B 0,C 180,E1 -10898.767,E2 -10898.767} C_VEL
LIN {X 0,Y 403.652,Z 594.862,A -85,B 0,C 180,E1 -10900.28,E2 -10900.28} C_VEL
LIN {X 0,Y 404.106,Z 586.188,A -85,B 0,C 180,E1 -10901.791,E2 -10901.791} C_VEL
LIN {X 0,Y 404.715,Z 577.293,A -85,B 0,C 180,E1 -10903.047,E2 -10903.047} C_VEL
LIN {X 0,Y 405.281,Z 568.759,A -85,B 0,C 180,E1 -10904.05,E2 -10904.05} C_VEL
LIN {X 0,Y 406.127,Z 556.984,A -85,B 0,C 180,E1 -10905.173,E2 -10905.173} C_VEL
LIN {X 0,Y 406.784,Z 547.184,A -85,B 0,C 180,E1 -10905.918,E2 -10905.918} C_VEL
LIN {X 0,Y 406.08,Z 535.748,A -85,B 0,C 180,E1 -10906.648,E2 -10906.648} C_VEL
LIN {X 0,Y 405.211,Z 522.535,A -85,B 0,C 180,E1 -10907.281,E2 -10907.281} C_VEL
LIN {X 0,Y 403.781,Z 508.874,A -85,B 0,C 180,E1 -10907.733,E2 -10907.733} C_VEL
LIN {X 0,Y 403.691,Z 507.394,A -85,B 0,C 180,E1 -10907.77,E2 -10907.77} C_VEL
LIN {X 0,Y 404.021,Z 495.921,A -85,B 0,C 180,E1 -10910.891,E2 -10910.891} C_VEL
LIN {X 0,Y 404.61,Z 482.158,A -85,B 0,C 180,E1 -10914.637,E2 -10914.637} C_VEL
LIN {X 0,Y 405.246,Z 469.155,A -85,B 0,C 180,E1 -10918.202,E2 -10918.202} C_VEL
LIN {X 0,Y 405.89,Z 459.089,A -85,B 0,C 180,E1 -10921.006,E2 -10921.006} C_VEL
LIN {X 0,Y 406.814,Z 445.935,A -85,B 0,C 180,E1 -10924.757,E2 -10924.757} C_VEL
LIN {X 0,Y 407.371,Z 438.864,A -85,B 0,C 180,E1 -10926.835,E2 -10926.835} C_VEL
LIN {X 0,Y 406.382,Z 432.362,A -85,B 0,C 180,E1 -10928.901,E2 -10928.901} C_VEL
LIN {X 0,Y 404.786,Z 423.996,A -85,B 0,C 180,E1 -10931.705,E2 -10931.705} C_VEL
LIN {X 0,Y 404.161,Z 421.144,A -85,B 0,C 180,E1 -10932.749,E2 -10932.749} C_VEL
LIN {X 0,Y 404.153,Z 421.144,A -85,B 0,C 180,E1 -10935.927,E2 -10935.927} C_VEL
LIN {X 0,Y 404.121,Z 421.147,A -85,B 0,C 180,E1 -10938.635,E2 -10938.635} C_VEL
LIN {X 0,Y 404.159,Z 421.14,A -85,B 0,C 180,E1 -10941.491,E2 -10941.491} C_VEL
LIN {X 0,Y 404.186,Z 421.136,A -85,B 0,C 180,E1 -10944.984,E2 -10944.984} C_VEL
LIN {X 0,Y 404.143,Z 421.144,A -85,B 0,C 180,E1 -10948.554,E2 -10948.554} C_VEL
LIN {X 0,Y 404.196,Z 421.139,A -85,B 0,C 180,E1 -10952,E2 -10952} C_VEL
LIN {X 0,Y 404.178,Z 421.137,A -85,B 0,C 180,E1 -10955.334,E2 -10955.334} C_VEL
LIN {X 0,Y 404.14,Z 421.144,A -85,B 0,C 180,E1 -10958.581,E2 -10958.581} C_VEL
LIN {X 0,Y 404.211,Z 421.135,A -85,B 0,C 180,E1 -10961.762,E2 -10961.762} C_VEL
LIN {X 0,Y 404.209,Z 421.133,A -85,B 0,C 180,E1 -10964.882,E2 -10964.882} C_VEL
LIN {X 0,Y 404.271,Z 421.13,A -85,B 0,C 180,E1 -10967.959,E2 -10967.959} C_VEL
LIN {X 0,Y 404.271,Z 421.125,A -85,B 0,C 180,E1 -10970.999,E2 -10970.999} C_VEL
LIN {X 0,Y 404.42,Z 421.112,A -85,B 0,C 180,E1 -10974.015,E2 -10974.015} C_VEL
LIN {X 0,Y 404.485,Z 421.104,A -85,B 0,C 180,E1 -10978.009,E2 -10978.009} C_VEL
LIN {X 0,Y 404.613,Z 421.087,A -85,B 0,C 180,E1 -10980,E2 -10980} C_VEL
LIN {X 0,Y 404.417,Z 421.107,A -85,B 0,C 180,E1 -10982.989,E2 -10982.989} C_VEL
LIN {X 0,Y 404.413,Z 421.107,A -85,B 0,C 180,E1 -10986.987,E2 -10986.987} C_VEL
LIN {X 0,Y 404.261,Z 421.132,A -85,B 0,C 180,E1 -10990.012,E2 -10990.012} C_VEL
LIN {X 0,Y 404.268,Z 421.126,A -85,B 0,C 180,E1 -10993.212,E2 -10993.212} C_VEL
LIN {X 0,Y 404.217,Z 421.131,A -85,B 0,C 180,E1 -10997.007,E2 -10997.007} C_VEL
LIN {X 0,Y 404.165,Z 421.141,A -85,B 0,C 180,E1 -11000.352,E2 -11000.352} C_VEL
LIN {X 0,Y 404.171,Z 421.141,A -85,B 0,C 180,E1 -11003.575,E2 -11003.575} C_VEL
LIN {X 0,Y 404.185,Z 421.14,A -85,B 0,C 180,E1 -11005.767,E2 -11005.767} C_VEL
LIN {X 0,Y 404.197,Z 421.139,A -85,B 0,C 180,E1 -11008,E2 -11008} C_VEL
LIN {X 0,Y 404.141,Z 421.144,A -85,B 0,C 180,E1 -11011.558,E2 -11011.558} C_VEL
LIN {X 0,Y 404.188,Z 421.136,A -85,B 0,C 180,E1 -11015.016,E2 -11015.016} C_VEL
LIN {X 0,Y 404.16,Z 421.139,A -85,B 0,C 180,E1 -11018.757,E2 -11018.757} C_VEL
LIN {X 0,Y 404.127,Z 421.147,A -85,B 0,C 180,E1 -11021.6,E2 -11021.6} C_VEL
LIN {X 0,Y 404.153,Z 421.141,A -85,B 0,C 180,E1 -11024.523,E2 -11024.523} C_VEL
LIN {X 0,Y 404.142,Z 421.143,A -85,B 0,C 180,E1 -11027.296,E2 -11027.296} C_VEL
LIN {X 0,Y 404.171,Z 421.142,A -85,B 0,C 180,E1 -11029.956,E2 -11029.956} C_VEL
LIN {X 0,Y 404.142,Z 421.142,A -85,B 0,C 180,E1 -11033.125,E2 -11033.125} C_VEL
LIN {X 0,Y 404.148,Z 421.143,A -85,B 0,C 180,E1 -11036.188,E2 -11036.188} C_VEL
LIN {X 0,Y 404.158,Z 421.144,A -85,B 0,C 180,E1 -11039.716,E2 -11039.716} C_VEL
LIN {X 0,Y 404.199,Z 421.135,A -85,B 0,C 180,E1 -11043.123,E2 -11043.123} C_VEL
LIN {X 0,Y 404.181,Z 421.139,A -85,B 0,C 180,E1 -11045.335,E2 -11045.335} C_VEL
LIN {X 0,Y 404.143,Z 421.141,A -85,B 0,C 180,E1 -11048.581,E2 -11048.581} C_VEL
LIN {X 0,Y 404.214,Z 421.137,A -85,B 0,C 180,E1 -11051.762,E2 -11051.762} C_VEL
LIN {X 0,Y 404.21,Z 421.137,A -85,B 0,C 180,E1 -11054.882,E2 -11054.882} C_VEL
LIN {X 0,Y 404.233,Z 421.135,A -85,B 0,C 180,E1 -11056.214,E2 -11056.214} C_VEL
LIN {X 0,Y 407.536,Z 432.235,A -85,B 0,C 180,E1 -11057.045,E2 -11057.045} C_VEL
LIN {X 0,Y 408.8,Z 437.113,A -85,B 0,C 180,E1 -11057.465,E2 -11057.465} C_VEL
LIN {X 0,Y 408.181,Z 448.596,A -85,B 0,C 180,E1 -11058.454,E2 -11058.454} C_VEL
LIN {X 0,Y 407.503,Z 458.745,A -85,B 0,C 180,E1 -11059.549,E2 -11059.549} C_VEL
LIN {X 0,Y 406.76,Z 468.189,A -85,B 0,C 180,E1 -11060.804,E2 -11060.804} C_VEL
LIN {X 0,Y 406.126,Z 477.091,A -85,B 0,C 180,E1 -11062.293,E2 -11062.293} C_VEL
LIN {X 0,Y 405.468,Z 484.275,A -85,B 0,C 180,E1 -11063.781,E2 -11063.781} C_VEL
LIN {X 0,Y 404.964,Z 490.857,A -85,B 0,C 180,E1 -11065.521,E2 -11065.521} C_VEL
LIN {X 0,Y 404.595,Z 495.205,A -85,B 0,C 180,E1 -11067.013,E2 -11067.013} C_VEL
LIN {X 0,Y 404.381,Z 497.503,A -85,B 0,C 180,E1 -11068.008,E2 -11068.008} C_VEL
LIN {X 0,Y 404.22,Z 499.384,A -85,B 0,C 180,E1 -11069.004,E2 -11069.004} C_VEL
LIN {X 0,Y 404.137,Z 500.853,A -85,B 0,C 180,E1 -11070,E2 -11070} C_VEL
LIN {X 0,Y 404.029,Z 502.545,A -85,B 0,C 180,E1 -11071.994,E2 -11071.994} C_VEL
LIN {X 0,Y 403.909,Z 502.849,A -85,B 0,C 180,E1 -11072.992,E2 -11072.992} C_VEL
LIN {X 0,Y 403.975,Z 502.756,A -85,B 0,C 180,E1 -11073.991,E2 -11073.991} C_VEL
LIN {X 0,Y 404.307,Z 501.333,A -85,B 0,C 180,E1 -11075.987,E2 -11075.987} C_VEL
LIN {X 0,Y 404.39,Z 500.068,A -85,B 0,C 180,E1 -11076.988,E2 -11076.988} C_VEL
LIN {X 0,Y 404.68,Z 497.362,A -85,B 0,C 180,E1 -11078.489,E2 -11078.489} C_VEL
LIN {X 0,Y 405.104,Z 493.645,A -85,B 0,C 180,E1 -11079.991,E2 -11079.991} C_VEL
LIN {X 0,Y 405.59,Z 488.652,A -85,B 0,C 180,E1 -11081.54,E2 -11081.54} C_VEL
LIN {X 0,Y 406.061,Z 482.746,A -85,B 0,C 180,E1 -11083.003,E2 -11083.003} C_VEL
LIN {X 0,Y 406.67,Z 475.924,A -85,B 0,C 180,E1 -11084.365,E2 -11084.365} C_VEL
LIN {X 0,Y 407.104,Z 471.514,A -85,B 0,C 180,E1 -11085.111,E2 -11085.111} C_VEL
LIN {X 0,Y 406.779,Z 467.69,A -85,B 0,C 180,E1 -11085.736,E2 -11085.736} C_VEL
LIN {X 0,Y 403.493,Z 458.699,A -85,B 0,C 180,E1 -11087.159,E2 -11087.159} C_VEL
LIN {X 0,Y 402.099,Z 452.98,A -85,B 0,C 180,E1 -11087.906,E2 -11087.906} C_VEL
LIN {X 0,Y 402.065,Z 449.775,A -85,B 0,C 180,E1 -11088.244,E2 -11088.244} C_VEL
LIN {X 0,Y 402.664,Z 439.876,A -85,B 0,C 180,E1 -11089.126,E2 -11089.126} C_VEL
LIN {X 0,Y 399.815,Z 430.131,A -85,B 0,C 180,E1 -11090.012,E2 -11090.012} C_VEL
LIN {X 0,Y 397.116,Z 422.02,A -85,B 0,C 180,E1 -11090.683,E2 -11090.683} C_VEL
LIN {X 0,Y 397.133,Z 422.016,A -85,B 0,C 180,E1 -11094.019,E2 -11094.019} C_VEL
LIN {X 0,Y 397.199,Z 422.004,A -85,B 0,C 180,E1 -11097.39,E2 -11097.39} C_VEL
LIN {X 0,Y 397.083,Z 422.02,A -85,B 0,C 180,E1 -11100.882,E2 -11100.882} C_VEL
LIN {X 0,Y 397.13,Z 422.016,A -85,B 0,C 180,E1 -11104.493,E2 -11104.493} C_VEL
LIN {X 0,Y 397.107,Z 422.021,A -85,B 0,C 180,E1 -11108.275,E2 -11108.275} C_VEL
LIN {X 0,Y 397.093,Z 422.018,A -85,B 0,C 180,E1 -11110.909,E2 -11110.909} C_VEL
LIN {X 0,Y 397.105,Z 422.018,A -85,B 0,C 180,E1 -11113.648,E2 -11113.648} C_VEL
LIN {X 0,Y 397.107,Z 422.018,A -85,B 0,C 180,E1 -11116.521,E2 -11116.521} C_VEL
LIN {X 0,Y 397.118,Z 422.017,A -85,B 0,C 180,E1 -11120.423,E2 -11120.423} C_VEL
LIN {X 0,Y 397.112,Z 422.018,A -85,B 0,C 180,E1 -11124.265,E2 -11124.265} C_VEL
LIN {X 0,Y 397.119,Z 422.014,A -85,B 0,C 180,E1 -11126.727,E2 -11126.727} C_VEL
LIN {X 0,Y 397.129,Z 422.015,A -85,B 0,C 180,E1 -11130.296,E2 -11130.296} C_VEL
LIN {X 0,Y 397.198,Z 422.005,A -85,B 0,C 180,E1 -11132.61,E2 -11132.61} C_VEL
LIN {X 0,Y 397.133,Z 422.017,A -85,B 0,C 180,E1 -11135.981,E2 -11135.981} C_VEL
LIN {X 0,Y 397.143,Z 422.018,A -85,B 0,C 180,E1 -11139.705,E2 -11139.705} C_VEL
LIN {X 0,Y 397.186,Z 422.006,A -85,B 0,C 180,E1 -11142.845,E2 -11142.845} C_VEL
LIN {X 0,Y 397.223,Z 422.001,A -85,B 0,C 180,E1 -11144.641,E2 -11144.641} C_VEL
LIN {X 0,Y 400.454,Z 434.585,A -85,B 0,C 180,E1 -11145.636,E2 -11145.636} C_VEL
LIN {X 0,Y 400.442,Z 442.465,A -85,B 0,C 180,E1 -11146.294,E2 -11146.294} C_VEL
LIN {X 0,Y 399.711,Z 453.903,A -85,B 0,C 180,E1 -11147.432,E2 -11147.432} C_VEL
LIN {X 0,Y 399.325,Z 463.263,A -85,B 0,C 180,E1 -11148.58,E2 -11148.58} C_VEL
LIN {X 0,Y 398.724,Z 471.924,A -85,B 0,C 180,E1 -11149.848,E2 -11149.848} C_VEL
LIN {X 0,Y 398.199,Z 479.811,A -85,B 0,C 180,E1 -11151.256,E2 -11151.256} C_VEL
LIN {X 0,Y 397.772,Z 487.225,A -85,B 0,C 180,E1 -11152.895,E2 -11152.895} C_VEL
LIN {X 0,Y 397.469,Z 492.729,A -85,B 0,C 180,E1 -11154.419,E2 -11154.419} C_VEL
LIN {X 0,Y 397.076,Z 497.071,A -85,B 0,C 180,E1 -11155.94,E2 -11155.94} C_VEL
LIN {X 0,Y 396.929,Z 499.34,A -85,B 0,C 180,E1 -11156.955,E2 -11156.955} C_VEL
LIN {X 0,Y 397.025,Z 501.143,A -85,B 0,C 180,E1 -11157.971,E2 -11157.971} C_VEL
LIN {X 0,Y 396.935,Z 502.576,A -85,B 0,C 180,E1 -11158.985,E2 -11158.985} C_VEL
LIN {X 0,Y 397.025,Z 503.542,A -85,B 0,C 180,E1 -11160,E2 -11160} C_VEL
LIN {X 0,Y 397.17,Z 504.291,A -85,B 0,C 180,E1 -11162.028,E2 -11162.028} C_VEL
LIN {X 0,Y 397.204,Z 504.077,A -85,B 0,C 180,E1 -11163.043,E2 -11163.043} C_VEL
LIN {X 0,Y 397.42,Z 502.38,A -85,B 0,C 180,E1 -11165.073,E2 -11165.073} C_VEL
LIN {X 0,Y 397.669,Z 500.917,A -85,B 0,C 180,E1 -11166.087,E2 -11166.087} C_VEL
LIN {X 0,Y 398.207,Z 497.839,A -85,B 0,C 180,E1 -11167.606,E2 -11167.606} C_VEL
LIN {X 0,Y 398.678,Z 493.538,A -85,B 0,C 180,E1 -11169.18,E2 -11169.18} C_VEL
LIN {X 0,Y 399.376,Z 487.381,A -85,B 0,C 180,E1 -11170.904,E2 -11170.904} C_VEL
LIN {X 0,Y 400.192,Z 480.457,A -85,B 0,C 180,E1 -11172.423,E2 -11172.423} C_VEL
LIN {X 0,Y 401.094,Z 471.755,A -85,B 0,C 180,E1 -11173.941,E2 -11173.941} C_VEL
LIN {X 0,Y 401.914,Z 462.837,A -85,B 0,C 180,E1 -11175.206,E2 -11175.206} C_VEL
LIN {X 0,Y 402.838,Z 452.789,A -85,B 0,C 180,E1 -11176.352,E2 -11176.352} C_VEL
LIN {X 0,Y 403.75,Z 440.747,A -85,B 0,C 180,E1 -11177.465,E2 -11177.465} C_VEL
LIN {X 0,Y 400.294,Z 430.174,A -85,B 0,C 180,E1 -11178.542,E2 -11178.542} C_VEL
LIN {X 0,Y 397.139,Z 422.025,A -85,B 0,C 180,E1 -11179.311,E2 -11179.311} C_VEL
LIN {X 0,Y 397.138,Z 422.019,A -85,B 0,C 180,E1 -11183.04,E2 -11183.04} C_VEL
LIN {X 0,Y 397.138,Z 422.016,A -85,B 0,C 180,E1 -11186.258,E2 -11186.258} C_VEL
LIN {X 0,Y 397.126,Z 422.019,A -85,B 0,C 180,E1 -11188.543,E2 -11188.543} C_VEL
LIN {X 0,Y 397.081,Z 422.023,A -85,B 0,C 180,E1 -11192.071,E2 -11192.071} C_VEL
LIN {X 0,Y 397.122,Z 422.017,A -85,B 0,C 180,E1 -11195.503,E2 -11195.503} C_VEL
LIN {X 0,Y 397.132,Z 422.017,A -85,B 0,C 180,E1 -11198.861,E2 -11198.861} C_VEL
LIN {X 0,Y 397.072,Z 422.023,A -85,B 0,C 180,E1 -11202.267,E2 -11202.267} C_VEL
LIN {X 0,Y 397.102,Z 422.019,A -85,B 0,C 180,E1 -11205.733,E2 -11205.733} C_VEL
LIN {X 0,Y 397.133,Z 422.159,A -85,B 0,C 180,E1 -11206.065,E2 -11206.065} C_VEL
LIN {X 0,Y 398.939,Z 430.828,A -85,B 0,C 180,E1 -11209.246,E2 -11209.246} C_VEL
LIN {X 0,Y 400.523,Z 439.273,A -85,B 0,C 180,E1 -11212.15,E2 -11212.15} C_VEL
LIN {X 0,Y 400.721,Z 443.138,A -85,B 0,C 180,E1 -11213.394,E2 -11213.394} C_VEL
LIN {X 0,Y 399.474,Z 456.284,A -85,B 0,C 180,E1 -11217.349,E2 -11217.349} C_VEL
LIN {X 0,Y 398.525,Z 468.774,A -85,B 0,C 180,E1 -11220.99,E2 -11220.99} C_VEL
LIN {X 0,Y 397.768,Z 481.418,A -85,B 0,C 180,E1 -11224.598,E2 -11224.598} C_VEL
LIN {X 0,Y 397.11,Z 494.141,A -85,B 0,C 180,E1 -11228.182,E2 -11228.182} C_VEL
LIN {X 0,Y 396.688,Z 505.679,A -85,B 0,C 180,E1 -11231.436,E2 -11231.436} C_VEL
LIN {X 0,Y 397.934,Z 515.214,A -85,B 0,C 180,E1 -11231.815,E2 -11231.815} C_VEL
LIN {X 0,Y 399.186,Z 527.488,A -85,B 0,C 180,E1 -11232.347,E2 -11232.347} C_VEL
LIN {X 0,Y 399.759,Z 540.147,A -85,B 0,C 180,E1 -11233.071,E2 -11233.071} C_VEL
LIN {X 0,Y 400.058,Z 550.302,A -85,B 0,C 180,E1 -11233.806,E2 -11233.806} C_VEL
LIN {X 0,Y 399.068,Z 561.897,A -85,B 0,C 180,E1 -11234.813,E2 -11234.813} C_VEL
LIN {X 0,Y 398.202,Z 572.372,A -85,B 0,C 180,E1 -11235.952,E2 -11235.952} C_VEL
LIN {X 0,Y 397.715,Z 578.296,A -85,B 0,C 180,E1 -11236.719,E2 -11236.719} C_VEL
LIN {X 0,Y 397.08,Z 586.737,A -85,B 0,C 180,E1 -11237.997,E2 -11237.997} C_VEL
LIN {X 0,Y 396.57,Z 595.049,A -85,B 0,C 180,E1 -11239.534,E2 -11239.534} C_VEL
LIN {X 0,Y 396.348,Z 601.786,A -85,B 0,C 180,E1 -11241.074,E2 -11241.074} C_VEL
LIN {X 0,Y 396.29,Z 607.943,A -85,B 0,C 180,E1 -11242.869,E2 -11242.869} C_VEL
LIN {X 0,Y 396.347,Z 611.975,A -85,B 0,C 180,E1 -11244.403,E2 -11244.403} C_VEL
LIN {X 0,Y 396.561,Z 614.973,A -85,B 0,C 180,E1 -11245.935,E2 -11245.935} C_VEL
LIN {X 0,Y 396.559,Z 617.381,A -85,B 0,C 180,E1 -11247.969,E2 -11247.969} C_VEL
LIN {X 0,Y 396.819,Z 618.016,A -85,B 0,C 180,E1 -11248.985,E2 -11248.985} C_VEL
LIN {X 0,Y 396.839,Z 618.175,A -85,B 0,C 180,E1 -11250,E2 -11250} C_VEL
LIN {X 0,Y 396.822,Z 617.91,A -85,B 0,C 180,E1 -11251.015,E2 -11251.015} C_VEL
LIN {X 0,Y 396.546,Z 616.136,A -85,B 0,C 180,E1 -11253.048,E2 -11253.048} C_VEL
LIN {X 0,Y 396.566,Z 614.612,A -85,B 0,C 180,E1 -11254.065,E2 -11254.065} C_VEL
LIN {X 0,Y 396.381,Z 611.461,A -85,B 0,C 180,E1 -11255.596,E2 -11255.596} C_VEL
LIN {X 0,Y 396.317,Z 607.231,A -85,B 0,C 180,E1 -11257.13,E2 -11257.13} C_VEL
LIN {X 0,Y 396.387,Z 600.76,A -85,B 0,C 180,E1 -11258.925,E2 -11258.925} C_VEL
LIN {X 0,Y 396.594,Z 593.736,A -85,B 0,C 180,E1 -11260.465,E2 -11260.465} C_VEL
LIN {X 0,Y 397.005,Z 586.609,A -85,B 0,C 180,E1 -11261.746,E2 -11261.746} C_VEL
LIN {X 0,Y 397.638,Z 578.063,A -85,B 0,C 180,E1 -11263.023,E2 -11263.023} C_VEL
LIN {X 0,Y 397.967,Z 571.83,A -85,B 0,C 180,E1 -11263.813,E2 -11263.813} C_VEL
LIN {X 0,Y 398.789,Z 561.316,A -85,B 0,C 180,E1 -11264.936,E2 -11264.936} C_VEL
LIN {X 0,Y 399.681,Z 549.442,A -85,B 0,C 180,E1 -11265.947,E2 -11265.947} C_VEL
LIN {X 0,Y 399.171,Z 537.028,A -85,B 0,C 180,E1 -11266.792,E2 -11266.792} C_VEL
LIN {X 0,Y 398.373,Z 523.93,A -85,B 0,C 180,E1 -11267.469,E2 -11267.469} C_VEL
LIN {X 0,Y 397.138,Z 510.985,A -85,B 0,C 180,E1 -11267.95,E2 -11267.95} C_VEL
LIN {X 0,Y 396.61,Z 506.304,A -85,B 0,C 180,E1 -11268.085,E2 -11268.085} C_VEL
LIN {X 0,Y 396.983,Z 494.854,A -85,B 0,C 180,E1 -11271.28,E2 -11271.28} C_VEL
LIN {X 0,Y 397.63,Z 481.132,A -85,B 0,C 180,E1 -11275.099,E2 -11275.099} C_VEL
LIN {X 0,Y 398.382,Z 467.167,A -85,B 0,C 180,E1 -11279.021,E2 -11279.021} C_VEL
LIN {X 0,Y 399.038,Z 457.116,A -85,B 0,C 180,E1 -11281.895,E2 -11281.895} C_VEL
LIN {X 0,Y 399.979,Z 445.012,A -85,B 0,C 180,E1 -11285.439,E2 -11285.439} C_VEL
LIN {X 0,Y 400.379,Z 439.207,A -85,B 0,C 180,E1 -11287.191,E2 -11287.191} C_VEL
LIN {X 0,Y 398.864,Z 430.691,A -85,B 0,C 180,E1 -11289.998,E2 -11289.998} C_VEL
LIN {X 0,Y 397.127,Z 422.022,A -85,B 0,C 180,E1 -11293.039,E2 -11293.039} C_VEL
LIN {X 0,Y 397.105,Z 422.024,A -85,B 0,C 180,E1 -11296.52,E2 -11296.52} C_VEL
LIN {X 0,Y 397.115,Z 422.021,A -85,B 0,C 180,E1 -11300.423,E2 -11300.423} C_VEL
LIN {X 0,Y 397.11,Z 422.022,A -85,B 0,C 180,E1 -11304.265,E2 -11304.265} C_VEL
LIN {X 0,Y 397.115,Z 422.018,A -85,B 0,C 180,E1 -11306.727,E2 -11306.727} C_VEL
LIN {X 0,Y 397.125,Z 422.02,A -85,B 0,C 180,E1 -11310.296,E2 -11310.296} C_VEL
LIN {X 0,Y 397.195,Z 422.009,A -85,B 0,C 180,E1 -11312.61,E2 -11312.61} C_VEL
LIN {X 0,Y 397.134,Z 422.019,A -85,B 0,C 180,E1 -11315.982,E2 -11315.982} C_VEL
LIN {X 0,Y 397.139,Z 422.015,A -85,B 0,C 180,E1 -11319.705,E2 -11319.705} C_VEL
LIN {X 0,Y 397.183,Z 422.009,A -85,B 0,C 180,E1 -11322.845,E2 -11322.845} C_VEL
LIN {X 0,Y 397.227,Z 422.004,A -85,B 0,C 180,E1 -11326.679,E2 -11326.679} C_VEL
LIN {X 0,Y 397.229,Z 422.006,A -85,B 0,C 180,E1 -11329.809,E2 -11329.809} C_VEL
LIN {X 0,Y 397.339,Z 421.988,A -85,B 0,C 180,E1 -11332.888,E2 -11332.888} C_VEL
LIN {X 0,Y 397.257,Z 421.999,A -85,B 0,C 180,E1 -11334.925,E2 -11334.925} C_VEL
LIN {X 0,Y 397.454,Z 421.979,A -85,B 0,C 180,E1 -11337.973,E2 -11337.973} C_VEL
LIN {X 0,Y 397.583,Z 421.963,A -85,B 0,C 180,E1 -11340,E2 -11340} C_VEL
LIN {X 0,Y 397.377,Z 421.983,A -85,B 0,C 180,E1 -11343.042,E2 -11343.042} C_VEL
LIN {X 0,Y 397.365,Z 421.985,A -85,B 0,C 180,E1 -11347.112,E2 -11347.112} C_VEL
LIN {X 0,Y 397.22,Z 422.008,A -85,B 0,C 180,E1 -11350.191,E2 -11350.191} C_VEL
LIN {X 0,Y 397.228,Z 422.003,A -85,B 0,C 180,E1 -11353.321,E2 -11353.321} C_VEL
LIN {X 0,Y 397.183,Z 422.008,A -85,B 0,C 180,E1 -11357.155,E2 -11357.155} C_VEL
LIN {X 0,Y 397.104,Z 422.018,A -85,B 0,C 180,E1 -11360.73,E2 -11360.73} C_VEL
LIN {X 0,Y 397.135,Z 422.019,A -85,B 0,C 180,E1 -11364.018,E2 -11364.018} C_VEL
LIN {X 0,Y 397.196,Z 422.008,A -85,B 0,C 180,E1 -11367.39,E2 -11367.39} C_VEL
LIN {X 0,Y 397.08,Z 422.021,A -85,B 0,C 180,E1 -11370.883,E2 -11370.883} C_VEL
LIN {X 0,Y 397.128,Z 422.016,A -85,B 0,C 180,E1 -11374.493,E2 -11374.493} C_VEL
LIN {X 0,Y 397.108,Z 422.02,A -85,B 0,C 180,E1 -11378.275,E2 -11378.275} C_VEL
LIN {X 0,Y 397.091,Z 422.019,A -85,B 0,C 180,E1 -11380.909,E2 -11380.909} C_VEL
LIN {X 0,Y 397.106,Z 422.022,A -85,B 0,C 180,E1 -11383.648,E2 -11383.648} C_VEL
LIN {X 0,Y 397.107,Z 422.018,A -85,B 0,C 180,E1 -11386.521,E2 -11386.521} C_VEL
LIN {X 0,Y 397.117,Z 422.017,A -85,B 0,C 180,E1 -11390.423,E2 -11390.423} C_VEL
LIN {X 0,Y 397.112,Z 422.018,A -85,B 0,C 180,E1 -11394.266,E2 -11394.266} C_VEL
LIN {X 0,Y 397.118,Z 422.016,A -85,B 0,C 180,E1 -11396.728,E2 -11396.728} C_VEL
LIN {X 0,Y 397.137,Z 422.015,A -85,B 0,C 180,E1 -11400.297,E2 -11400.297} C_VEL
LIN {X 0,Y 397.198,Z 422.006,A -85,B 0,C 180,E1 -11402.61,E2 -11402.61} C_VEL
LIN {X 0,Y 397.137,Z 422.017,A -85,B 0,C 180,E1 -11405.982,E2 -11405.982} C_VEL
LIN {X 0,Y 397.142,Z 422.018,A -85,B 0,C 180,E1 -11409.705,E2 -11409.705} C_VEL
LIN {X 0,Y 397.186,Z 422.008,A -85,B 0,C 180,E1 -11412.845,E2 -11412.845} C_VEL
LIN {X 0,Y 397.179,Z 422.013,A -85,B 0,C 180,E1 -11415.919,E2 -11415.919} C_VEL
LIN {X 0,Y 400.72,Z 433.724,A -85,B 0,C 180,E1 -11416.821,E2 -11416.821} C_VEL
LIN {X 0,Y 401.986,Z 438.547,A -85,B 0,C 180,E1 -11417.249,E2 -11417.249} C_VEL
LIN {X 0,Y 401.33,Z 449.944,A -85,B 0,C 180,E1 -11418.254,E2 -11418.254} C_VEL
LIN {X 0,Y 400.625,Z 460.034,A -85,B 0,C 180,E1 -11419.367,E2 -11419.367} C_VEL
LIN {X 0,Y 399.853,Z 469.421,A -85,B 0,C 180,E1 -11420.643,E2 -11420.643} C_VEL
LIN {X 0,Y 399.19,Z 478.277,A -85,B 0,C 180,E1 -11422.158,E2 -11422.158} C_VEL
LIN {X 0,Y 398.512,Z 485.429,A -85,B 0,C 180,E1 -11423.672,E2 -11423.672} C_VEL
LIN {X 0,Y 397.973,Z 491.973,A -85,B 0,C 180,E1 -11425.442,E2 -11425.442} C_VEL
LIN {X 0,Y 397.592,Z 496.296,A -85,B 0,C 180,E1 -11426.96,E2 -11426.96} C_VEL
LIN {X 0,Y 397.368,Z 498.584,A -85,B 0,C 180,E1 -11427.973,E2 -11427.973} C_VEL
LIN {X 0,Y 397.201,Z 500.454,A -85,B 0,C 180,E1 -11428.986,E2 -11428.986} C_VEL
LIN {X 0,Y 397.117,Z 501.905,A -85,B 0,C 180,E1 -11430,E2 -11430} C_VEL
LIN {X 0,Y 397.006,Z 503.572,A -85,B 0,C 180,E1 -11432.029,E2 -11432.029} C_VEL
LIN {X 0,Y 396.884,Z 503.867,A -85,B 0,C 180,E1 -11433.045,E2 -11433.045} C_VEL
LIN {X 0,Y 396.954,Z 503.758,A -85,B 0,C 180,E1 -11434.061,E2 -11434.061} C_VEL
LIN {X 0,Y 397.312,Z 502.308,A -85,B 0,C 180,E1 -11436.093,E2 -11436.093} C_VEL
LIN {X 0,Y 397.405,Z 501.033,A -85,B 0,C 180,E1 -11437.111,E2 -11437.111} C_VEL
LIN {X 0,Y 397.705,Z 498.307,A -85,B 0,C 180,E1 -11438.639,E2 -11438.639} C_VEL
LIN {X 0,Y 398.174,Z 494.564,A -85,B 0,C 180,E1 -11440.167,E2 -11440.167} C_VEL
LIN {X 0,Y 398.674,Z 489.716,A -85,B 0,C 180,E1 -11441.697,E2 -11441.697} C_VEL
LIN {X 0,Y 399.195,Z 483.61,A -85,B 0,C 180,E1 -11443.231,E2 -11443.231} C_VEL
LIN {X 0,Y 399.838,Z 476.835,A -85,B 0,C 180,E1 -11444.6,E2 -11444.6} C_VEL
LIN {X 0,Y 400.702,Z 468.019,A -85,B 0,C 180,E1 -11446.036,E2 -11446.036} C_VEL
LIN {X 0,Y 401.396,Z 458.374,A -85,B 0,C 180,E1 -11447.317,E2 -11447.317} C_VEL
LIN {X 0,Y 402.065,Z 449.775,A -85,B 0,C 180,E1 -11448.244,E2 -11448.244} C_VEL
LIN {X 0,Y 401.888,Z 446.603,A -85,B 0,C 180,E1 -11448.572,E2 -11448.572} C_VEL
LIN {X 0,Y 400.33,Z 442.099,A -85,B 0,C 180,E1 -11449.075,E2 -11449.075} C_VEL
LIN {X 0,Y 397.849,Z 437.865,A -85,B 0,C 180,E1 -11449.568,E2 -11449.568} C_VEL
LIN {X 0,Y 394.045,Z 432.114,A -85,B 0,C 180,E1 -11450.211,E2 -11450.211} C_VEL
LIN {X 0,Y 391.626,Z 427.422,A -85,B 0,C 180,E1 -11450.66,E2 -11450.66} C_VEL
LIN {X 0,Y 391.009,Z 425.731,A -85,B 0,C 180,E1 -11450.799,E2 -11450.799} C_VEL
LIN {X 0,Y 390.058,Z 422.898,A -85,B 0,C 180,E1 -11451.025,E2 -11451.025} C_VEL
LIN {X 0,Y 390.082,Z 422.896,A -85,B 0,C 180,E1 -11454.481,E2 -11454.481} C_VEL
LIN {X 0,Y 390.121,Z 422.889,A -85,B 0,C 180,E1 -11457.93,E2 -11457.93} C_VEL
LIN {X 0,Y 390.028,Z 422.898,A -85,B 0,C 180,E1 -11461.504,E2 -11461.504} C_VEL
LIN {X 0,Y 390.073,Z 422.897,A -85,B 0,C 180,E1 -11464.025,E2 -11464.025} C_VEL
LIN {X 0,Y 390.047,Z 422.896,A -85,B 0,C 180,E1 -11467.551,E2 -11467.551} C_VEL
LIN {X 0,Y 390.06,Z 422.894,A -85,B 0,C 180,E1 -11470.821,E2 -11470.821} C_VEL
LIN {X 0,Y 390.059,Z 422.898,A -85,B 0,C 180,E1 -11473.886,E2 -11473.886} C_VEL
LIN {X 0,Y 390.062,Z 422.894,A -85,B 0,C 180,E1 -11476.79,E2 -11476.79} C_VEL
LIN {X 0,Y 390.06,Z 422.896,A -85,B 0,C 180,E1 -11479.561,E2 -11479.561} C_VEL
LIN {X 0,Y 390.047,Z 422.897,A -85,B 0,C 180,E1 -11482.449,E2 -11482.449} C_VEL
LIN {X 0,Y 390.088,Z 422.896,A -85,B 0,C 180,E1 -11486.047,E2 -11486.047} C_VEL
LIN {X 0,Y 390.051,Z 422.902,A -85,B 0,C 180,E1 -11489.869,E2 -11489.869} C_VEL
LIN {X 0,Y 390.117,Z 422.887,A -85,B 0,C 180,E1 -11493.232,E2 -11493.232} C_VEL
LIN {X 0,Y 390.08,Z 422.891,A -85,B 0,C 180,E1 -11496.761,E2 -11496.761} C_VEL
LIN {X 0,Y 390.108,Z 422.892,A -85,B 0,C 180,E1 -11499.983,E2 -11499.983} C_VEL
LIN {X 0,Y 390.142,Z 422.885,A -85,B 0,C 180,E1 -11503.248,E2 -11503.248} C_VEL
LIN {X 0,Y 390.18,Z 422.879,A -85,B 0,C 180,E1 -11504.442,E2 -11504.442} C_VEL
LIN {X 0,Y 393.194,Z 434.659,A -85,B 0,C 180,E1 -11505.365,E2 -11505.365} C_VEL
LIN {X 0,Y 393.672,Z 438.076,A -85,B 0,C 180,E1 -11505.658,E2 -11505.658} C_VEL
LIN {X 0,Y 393.135,Z 449.396,A -85,B 0,C 180,E1 -11506.693,E2 -11506.693} C_VEL
LIN {X 0,Y 392.566,Z 459.709,A -85,B 0,C 180,E1 -11507.856,E2 -11507.856} C_VEL
LIN {X 0,Y 391.988,Z 469.154,A -85,B 0,C 180,E1 -11509.149,E2 -11509.149} C_VEL
LIN {X 0,Y 391.389,Z 478.336,A -85,B 0,C 180,E1 -11510.699,E2 -11510.699} C_VEL
LIN {X 0,Y 390.977,Z 485.781,A -85,B 0,C 180,E1 -11512.252,E2 -11512.252} C_VEL
LIN {X 0,Y 390.53,Z 491.801,A -85,B 0,C 180,E1 -11513.801,E2 -11513.801} C_VEL
LIN {X 0,Y 390.325,Z 496.548,A -85,B 0,C 180,E1 -11515.352,E2 -11515.352} C_VEL
LIN {X 0,Y 389.896,Z 500.237,A -85,B 0,C 180,E1 -11516.9,E2 -11516.9} C_VEL
LIN {X 0,Y 390.002,Z 502.073,A -85,B 0,C 180,E1 -11517.934,E2 -11517.934} C_VEL
LIN {X 0,Y 389.912,Z 503.548,A -85,B 0,C 180,E1 -11518.967,E2 -11518.967} C_VEL
LIN {X 0,Y 390.012,Z 504.57,A -85,B 0,C 180,E1 -11520,E2 -11520} C_VEL
LIN {X 0,Y 390.167,Z 505.386,A -85,B 0,C 180,E1 -11522.064,E2 -11522.064} C_VEL
LIN {X 0,Y 390.226,Z 505.215,A -85,B 0,C 180,E1 -11523.097,E2 -11523.097} C_VEL
LIN {X 0,Y 390.449,Z 503.582,A -85,B 0,C 180,E1 -11525.163,E2 -11525.163} C_VEL
LIN {X 0,Y 390.719,Z 502.159,A -85,B 0,C 180,E1 -11526.196,E2 -11526.196} C_VEL
LIN {X 0,Y 391.297,Z 499.16,A -85,B 0,C 180,E1 -11527.741,E2 -11527.741} C_VEL
LIN {X 0,Y 391.883,Z 494.556,A -85,B 0,C 180,E1 -11529.47,E2 -11529.47} C_VEL
LIN {X 0,Y 392.565,Z 488.873,A -85,B 0,C 180,E1 -11531.096,E2 -11531.096} C_VEL
LIN {X 0,Y 393.435,Z 482.033,A -85,B 0,C 180,E1 -11532.64,E2 -11532.64} C_VEL
LIN {X 0,Y 394.415,Z 473.439,A -85,B 0,C 180,E1 -11534.182,E2 -11534.182} C_VEL
LIN {X 0,Y 395.292,Z 464.711,A -85,B 0,C 180,E1 -11535.467,E2 -11535.467} C_VEL
LIN {X 0,Y 396.288,Z 454.938,A -85,B 0,C 180,E1 -11536.63,E2 -11536.63} C_VEL
LIN {X 0,Y 397.263,Z 442.795,A -85,B 0,C 180,E1 -11537.789,E2 -11537.789} C_VEL
LIN {X 0,Y 393.791,Z 432.143,A -85,B 0,C 180,E1 -11538.933,E2 -11538.933} C_VEL
LIN {X 0,Y 390.215,Z 423.51,A -85,B 0,C 180,E1 -11539.805,E2 -11539.805} C_VEL
LIN {X 0,Y 390.108,Z 422.899,A -85,B 0,C 180,E1 -11539.879,E2 -11539.879} C_VEL
LIN {X 0,Y 390.092,Z 422.897,A -85,B 0,C 180,E1 -11543.351,E2 -11543.351} C_VEL
LIN {X 0,Y 390.116,Z 422.892,A -85,B 0,C 180,E1 -11546.768,E2 -11546.768} C_VEL
LIN {X 0,Y 390.042,Z 422.901,A -85,B 0,C 180,E1 -11550.299,E2 -11550.299} C_VEL
LIN {X 0,Y 390.071,Z 422.896,A -85,B 0,C 180,E1 -11554.024,E2 -11554.024} C_VEL
LIN {X 0,Y 390.046,Z 422.898,A -85,B 0,C 180,E1 -11557.551,E2 -11557.551} C_VEL
LIN {X 0,Y 390.059,Z 422.898,A -85,B 0,C 180,E1 -11560.821,E2 -11560.821} C_VEL
LIN {X 0,Y 390.057,Z 422.895,A -85,B 0,C 180,E1 -11563.886,E2 -11563.886} C_VEL
LIN {X 0,Y 390.085,Z 423.088,A -85,B 0,C 180,E1 -11565.685,E2 -11565.685} C_VEL
LIN {X 0,Y 391.856,Z 431.6,A -85,B 0,C 180,E1 -11568.875,E2 -11568.875} C_VEL
LIN {X 0,Y 393.434,Z 439.907,A -85,B 0,C 180,E1 -11571.812,E2 -11571.812} C_VEL
LIN {X 0,Y 393.8,Z 443.822,A -85,B 0,C 180,E1 -11573.109,E2 -11573.109} C_VEL
LIN {X 0,Y 392.598,Z 456.006,A -85,B 0,C 180,E1 -11576.866,E2 -11576.866} C_VEL
LIN {X 0,Y 391.624,Z 467.929,A -85,B 0,C 180,E1 -11580.428,E2 -11580.428} C_VEL
LIN {X 0,Y 390.871,Z 479.205,A -85,B 0,C 180,E1 -11583.727,E2 -11583.727} C_VEL
LIN {X 0,Y 390.203,Z 491.314,A -85,B 0,C 180,E1 -11587.224,E2 -11587.224} C_VEL
LIN {X 0,Y 389.657,Z 504.119,A -85,B 0,C 180,E1 -11590.918,E2 -11590.918} C_VEL
LIN {X 0,Y 391.365,Z 518.171,A -85,B 0,C 180,E1 -11591.616,E2 -11591.616} C_VEL
LIN {X 0,Y 392.595,Z 531.628,A -85,B 0,C 180,E1 -11592.282,E2 -11592.282} C_VEL
LIN {X 0,Y 392.974,Z 544.291,A -85,B 0,C 180,E1 -11593.105,E2 -11593.105} C_VEL
LIN {X 0,Y 393.086,Z 551.122,A -85,B 0,C 180,E1 -11593.644,E2 -11593.644} C_VEL
LIN {X 0,Y 392.057,Z 562.378,A -85,B 0,C 180,E1 -11594.668,E2 -11594.668} C_VEL
LIN {X 0,Y 391.142,Z 572.73,A -85,B 0,C 180,E1 -11595.852,E2 -11595.852} C_VEL
LIN {X 0,Y 390.562,Z 580.99,A -85,B 0,C 180,E1 -11597.001,E2 -11597.001} C_VEL
LIN {X 0,Y 389.902,Z 588.799,A -85,B 0,C 180,E1 -11598.3,E2 -11598.3} C_VEL
LIN {X 0,Y 389.395,Z 596.496,A -85,B 0,C 180,E1 -11599.864,E2 -11599.864} C_VEL
LIN {X 0,Y 389.243,Z 601.798,A -85,B 0,C 180,E1 -11601.172,E2 -11601.172} C_VEL
LIN {X 0,Y 389.225,Z 606.971,A -85,B 0,C 180,E1 -11602.738,E2 -11602.738} C_VEL
LIN {X 0,Y 389.281,Z 610.992,A -85,B 0,C 180,E1 -11604.301,E2 -11604.301} C_VEL
LIN {X 0,Y 389.499,Z 613.979,A -85,B 0,C 180,E1 -11605.861,E2 -11605.861} C_VEL
LIN {X 0,Y 389.483,Z 615.381,A -85,B 0,C 180,E1 -11606.897,E2 -11606.897} C_VEL
LIN {X 0,Y 389.791,Z 617.011,A -85,B 0,C 180,E1 -11608.967,E2 -11608.967} C_VEL
LIN {X 0,Y 389.817,Z 617.161,A -85,B 0,C 180,E1 -11610,E2 -11610} C_VEL
LIN {X 0,Y 389.795,Z 616.888,A -85,B 0,C 180,E1 -11611.033,E2 -11611.033} C_VEL
LIN {X 0,Y 389.505,Z 615.099,A -85,B 0,C 180,E1 -11613.103,E2 -11613.103} C_VEL
LIN {X 0,Y 389.443,Z 612.62,A -85,B 0,C 180,E1 -11614.658,E2 -11614.658} C_VEL
LIN {X 0,Y 389.312,Z 609.098,A -85,B 0,C 180,E1 -11616.218,E2 -11616.218} C_VEL
LIN {X 0,Y 389.248,Z 604.464,A -85,B 0,C 180,E1 -11617.782,E2 -11617.782} C_VEL
LIN {X 0,Y 389.402,Z 597.478,A -85,B 0,C 180,E1 -11619.61,E2 -11619.61} C_VEL
LIN {X 0,Y 389.741,Z 589.897,A -85,B 0,C 180,E1 -11621.177,E2 -11621.177} C_VEL
LIN {X 0,Y 390.392,Z 580.533,A -85,B 0,C 180,E1 -11622.74,E2 -11622.74} C_VEL
LIN {X 0,Y 390.805,Z 572.744,A -85,B 0,C 180,E1 -11623.807,E2 -11623.807} C_VEL
LIN {X 0,Y 391.681,Z 562.707,A -85,B 0,C 180,E1 -11624.947,E2 -11624.947} C_VEL
LIN {X 0,Y 392.595,Z 551.385,A -85,B 0,C 180,E1 -11625.976,E2 -11625.976} C_VEL
LIN {X 0,Y 392.61,Z 546.294,A -85,B 0,C 180,E1 -11626.376,E2 -11626.376} C_VEL
LIN {X 0,Y 392.118,Z 534.489,A -85,B 0,C 180,E1 -11627.167,E2 -11627.167} C_VEL
LIN {X 0,Y 391.217,Z 521.245,A -85,B 0,C 180,E1 -11627.845,E2 -11627.845} C_VEL
LIN {X 0,Y 389.815,Z 507.842,A -85,B 0,C 180,E1 -11628.322,E2 -11628.322} C_VEL
LIN {X 0,Y 389.557,Z 505.302,A -85,B 0,C 180,E1 -11628.406,E2 -11628.406} C_VEL
LIN {X 0,Y 389.955,Z 493.785,A -85,B 0,C 180,E1 -11631.682,E2 -11631.682} C_VEL
LIN {X 0,Y 390.618,Z 480.097,A -85,B 0,C 180,E1 -11635.582,E2 -11635.582} C_VEL
LIN {X 0,Y 391.483,Z 466.178,A -85,B 0,C 180,E1 -11639.583,E2 -11639.583} C_VEL
LIN {X 0,Y 392.347,Z 454.143,A -85,B 0,C 180,E1 -11643.116,E2 -11643.116} C_VEL
LIN {X 0,Y 393.327,Z 442.988,A -85,B 0,C 180,E1 -11646.48,E2 -11646.48} C_VEL
LIN {X 0,Y 393.178,Z 438.976,A -85,B 0,C 180,E1 -11647.756,E2 -11647.756} C_VEL
LIN {X 0,Y 391.4,Z 429.32,A -85,B 0,C 180,E1 -11651.048,E2 -11651.048} C_VEL
LIN {X 0,Y 390.069,Z 422.899,A -85,B 0,C 180,E1 -11653.431,E2 -11653.431} C_VEL
LIN {X 0,Y 390.06,Z 422.905,A -85,B 0,C 180,E1 -11656.79,E2 -11656.79} C_VEL
LIN {X 0,Y 390.058,Z 422.896,A -85,B 0,C 180,E1 -11659.561,E2 -11659.561} C_VEL
LIN {X 0,Y 390.047,Z 422.901,A -85,B 0,C 180,E1 -11662.449,E2 -11662.449} C_VEL
LIN {X 0,Y 390.085,Z 422.897,A -85,B 0,C 180,E1 -11666.047,E2 -11666.047} C_VEL
LIN {X 0,Y 390.047,Z 422.9,A -85,B 0,C 180,E1 -11669.869,E2 -11669.869} C_VEL
LIN {X 0,Y 390.114,Z 422.888,A -85,B 0,C 180,E1 -11673.232,E2 -11673.232} C_VEL
LIN {X 0,Y 390.107,Z 422.89,A -85,B 0,C 180,E1 -11676.75,E2 -11676.75} C_VEL
LIN {X 0,Y 390.105,Z 422.894,A -85,B 0,C 180,E1 -11679.983,E2 -11679.983} C_VEL
LIN {X 0,Y 390.139,Z 422.885,A -85,B 0,C 180,E1 -11683.248,E2 -11683.248} C_VEL
LIN {X 0,Y 390.195,Z 422.88,A -85,B 0,C 180,E1 -11686.562,E2 -11686.562} C_VEL
LIN {X 0,Y 390.179,Z 422.882,A -85,B 0,C 180,E1 -11689.623,E2 -11689.623} C_VEL
LIN {X 0,Y 390.286,Z 422.867,A -85,B 0,C 180,E1 -11692.759,E2 -11692.759} C_VEL
LIN {X 0,Y 390.228,Z 422.874,A -85,B 0,C 180,E1 -11694.834,E2 -11694.834} C_VEL
LIN {X 0,Y 390.423,Z 422.855,A -85,B 0,C 180,E1 -11697.937,E2 -11697.937} C_VEL
LIN {X 0,Y 390.552,Z 422.839,A -85,B 0,C 180,E1 -11700,E2 -11700} C_VEL
LIN {X 0,Y 390.312,Z 422.863,A -85,B 0,C 180,E1 -11703.097,E2 -11703.097} C_VEL
LIN {X 0,Y 390.311,Z 422.865,A -85,B 0,C 180,E1 -11706.653,E2 -11706.653} C_VEL
LIN {X 0,Y 390.207,Z 422.878,A -85,B 0,C 180,E1 -11709.329,E2 -11709.329} C_VEL
LIN {X 0,Y 390.172,Z 422.883,A -85,B 0,C 180,E1 -11712.483,E2 -11712.483} C_VEL
LIN {X 0,Y 390.141,Z 422.888,A -85,B 0,C 180,E1 -11715.677,E2 -11715.677} C_VEL
LIN {X 0,Y 390.107,Z 422.889,A -85,B 0,C 180,E1 -11718.922,E2 -11718.922} C_VEL
LIN {X 0,Y 390.042,Z 422.901,A -85,B 0,C 180,E1 -11722.234,E2 -11722.234} C_VEL
LIN {X 0,Y 390.121,Z 422.892,A -85,B 0,C 180,E1 -11725.744,E2 -11725.744} C_VEL
LIN {X 0,Y 390.06,Z 422.895,A -85,B 0,C 180,E1 -11729.11,E2 -11729.11} C_VEL
LIN {X 0,Y 390.045,Z 422.897,A -85,B 0,C 180,E1 -11732.722,E2 -11732.722} C_VEL
LIN {X 0,Y 390.059,Z 422.9,A -85,B 0,C 180,E1 -11735.826,E2 -11735.826} C_VEL
LIN {X 0,Y 390.073,Z 422.894,A -85,B 0,C 180,E1 -11739.219,E2 -11739.219} C_VEL
LIN {X 0,Y 390.047,Z 422.898,A -85,B 0,C 180,E1 -11742.375,E2 -11742.375} C_VEL
LIN {X 0,Y 390.05,Z 422.898,A -85,B 0,C 180,E1 -11745.355,E2 -11745.355} C_VEL
LIN {X 0,Y 390.035,Z 422.901,A -85,B 0,C 180,E1 -11748.187,E2 -11748.187} C_VEL
LIN {X 0,Y 390.094,Z 422.891,A -85,B 0,C 180,E1 -11750.908,E2 -11750.908} C_VEL
LIN {X 0,Y 390.088,Z 422.891,A -85,B 0,C 180,E1 -11754.794,E2 -11754.794} C_VEL
LIN {X 0,Y 390.05,Z 422.897,A -85,B 0,C 180,E1 -11758.498,E2 -11758.498} C_VEL
LIN {X 0,Y 390.12,Z 422.891,A -85,B 0,C 180,E1 -11762.07,E2 -11762.07} C_VEL
LIN {X 0,Y 390.084,Z 422.896,A -85,B 0,C 180,E1 -11765.52,E2 -11765.52} C_VEL
LIN {X 0,Y 390.059,Z 422.895,A -85,B 0,C 180,E1 -11768.878,E2 -11768.878} C_VEL
LIN {X 0,Y 390.132,Z 422.888,A -85,B 0,C 180,E1 -11772.167,E2 -11772.167} C_VEL
LIN {X 0,Y 390.136,Z 422.891,A -85,B 0,C 180,E1 -11775.603,E2 -11775.603} C_VEL
LIN {X 0,Y 393.883,Z 435.198,A -85,B 0,C 180,E1 -11776.588,E2 -11776.588} C_VEL
LIN {X 0,Y 395.161,Z 439.969,A -85,B 0,C 180,E1 -11777.024,E2 -11777.024} C_VEL
LIN {X 0,Y 394.479,Z 451.289,A -85,B 0,C 180,E1 -11778.047,E2 -11778.047} C_VEL
LIN {X 0,Y 393.741,Z 461.322,A -85,B 0,C 180,E1 -11779.179,E2 -11779.179} C_VEL
LIN {X 0,Y 392.949,Z 470.646,A -85,B 0,C 180,E1 -11780.477,E2 -11780.477} C_VEL
LIN {X 0,Y 392.255,Z 479.462,A -85,B 0,C 180,E1 -11782.019,E2 -11782.019} C_VEL
LIN {X 0,Y 391.553,Z 486.583,A -85,B 0,C 180,E1 -11783.559,E2 -11783.559} C_VEL
LIN {X 0,Y 390.983,Z 493.088,A -85,B 0,C 180,E1 -11785.361,E2 -11785.361} C_VEL
LIN {X 0,Y 390.589,Z 497.387,A -85,B 0,C 180,E1 -11786.906,E2 -11786.906} C_VEL
LIN {X 0,Y 390.354,Z 499.664,A -85,B 0,C 180,E1 -11787.937,E2 -11787.937} C_VEL
LIN {X 0,Y 390.182,Z 501.523,A -85,B 0,C 180,E1 -11788.968,E2 -11788.968} C_VEL
LIN {X 0,Y 390.097,Z 502.953,A -85,B 0,C 180,E1 -11790,E2 -11790} C_VEL
LIN {X 0,Y 389.982,Z 504.6,A -85,B 0,C 180,E1 -11792.066,E2 -11792.066} C_VEL
LIN {X 0,Y 389.86,Z 504.885,A -85,B 0,C 180,E1 -11793.1,E2 -11793.1} C_VEL
LIN {X 0,Y 389.934,Z 504.757,A -85,B 0,C 180,E1 -11794.135,E2 -11794.135} C_VEL
LIN {X 0,Y 390.318,Z 503.283,A -85,B 0,C 180,E1 -11796.202,E2 -11796.202} C_VEL
LIN {X 0,Y 390.422,Z 501.998,A -85,B 0,C 180,E1 -11797.239,E2 -11797.239} C_VEL
LIN {X 0,Y 390.748,Z 499.25,A -85,B 0,C 180,E1 -11798.794,E2 -11798.794} C_VEL
LIN {X 0,Y 391.249,Z 495.483,A -85,B 0,C 180,E1 -11800.348,E2 -11800.348} C_VEL
LIN {X 0,Y 391.773,Z 490.612,A -85,B 0,C 180,E1 -11801.906,E2 -11801.906} C_VEL
LIN {X 0,Y 392.338,Z 484.473,A -85,B 0,C 180,E1 -11803.466,E2 -11803.466} C_VEL
LIN {X 0,Y 393.005,Z 477.774,A -85,B 0,C 180,E1 -11804.839,E2 -11804.839} C_VEL
LIN {X 0,Y 393.906,Z 468.802,A -85,B 0,C 180,E1 -11806.321,E2 -11806.321} C_VEL
LIN {X 0,Y 394.669,Z 459.108,A -85,B 0,C 180,E1 -11807.622,E2 -11807.622} C_VEL
LIN {X 0,Y 395.452,Z 449.53,A -85,B 0,C 180,E1 -11808.657,E2 -11808.657} C_VEL
LIN {X 0,Y 395.913,Z 441.618,A -85,B 0,C 180,E1 -11809.367,E2 -11809.367} C_VEL
LIN {X 0,Y 392.999,Z 431.663,A -85,B 0,C 180,E1 -11810.304,E2 -11810.304} C_VEL
LIN {X 0,Y 391.009,Z 425.731,A -85,B 0,C 180,E1 -11810.799,E2 -11810.799} C_VEL
LIN {X 0,Y 390.158,Z 424.088,A -85,B 0,C 180,E1 -11811.05,E2 -11811.05} C_VEL
LIN {X 0,Y 388.815,Z 423.165,A -85,B 0,C 180,E1 -11811.505,E2 -11811.505} C_VEL
LIN {X 0,Y 385.928,Z 423.411,A -85,B 0,C 180,E1 -11812.719,E2 -11812.719} C_VEL
LIN {X 0,Y 383.875,Z 423.819,A -85,B 0,C 180,E1 -11813.993,E2 -11813.993} C_VEL
LIN {X 0,Y 383.051,Z 423.767,A -85,B 0,C 180,E1 -11815.302,E2 -11815.302} C_VEL
LIN {X 0,Y 383.045,Z 423.772,A -85,B 0,C 180,E1 -11818.493,E2 -11818.493} C_VEL
LIN {X 0,Y 383.014,Z 423.777,A -85,B 0,C 180,E1 -11822.15,E2 -11822.15} C_VEL
LIN {X 0,Y 383.022,Z 423.772,A -85,B 0,C 180,E1 -11824.668,E2 -11824.668} C_VEL
LIN {X 0,Y 383.004,Z 423.776,A -85,B 0,C 180,E1 -11827.904,E2 -11827.904} C_VEL
LIN {X 0,Y 382.988,Z 423.775,A -85,B 0,C 180,E1 -11831.347,E2 -11831.347} C_VEL
LIN {X 0,Y 383.001,Z 423.777,A -85,B 0,C 180,E1 -11834.303,E2 -11834.303} C_VEL
LIN {X 0,Y 383.014,Z 423.772,A -85,B 0,C 180,E1 -11837.24,E2 -11837.24} C_VEL
LIN {X 0,Y 383.019,Z 423.773,A -85,B 0,C 180,E1 -11840.414,E2 -11840.414} C_VEL
LIN {X 0,Y 383.029,Z 423.775,A -85,B 0,C 180,E1 -11844.044,E2 -11844.044} C_VEL
LIN {X 0,Y 382.991,Z 423.777,A -85,B 0,C 180,E1 -11847.578,E2 -11847.578} C_VEL
LIN {X 0,Y 382.996,Z 423.776,A -85,B 0,C 180,E1 -11850.3,E2 -11850.3} C_VEL
LIN {X 0,Y 383.061,Z 423.766,A -85,B 0,C 180,E1 -11852.698,E2 -11852.698} C_VEL
LIN {X 0,Y 383.055,Z 423.767,A -85,B 0,C 180,E1 -11855.04,E2 -11855.04} C_VEL
LIN {X 0,Y 382.996,Z 423.774,A -85,B 0,C 180,E1 -11858.469,E2 -11858.469} C_VEL
LIN {X 0,Y 383.093,Z 423.767,A -85,B 0,C 180,E1 -11861.828,E2 -11861.828} C_VEL
LIN {X 0,Y 383.164,Z 423.938,A -85,B 0,C 180,E1 -11864.252,E2 -11864.252} C_VEL
LIN {X 0,Y 386.32,Z 436.269,A -85,B 0,C 180,E1 -11865.245,E2 -11865.245} C_VEL
LIN {X 0,Y 386.728,Z 437.979,A -85,B 0,C 180,E1 -11865.4,E2 -11865.4} C_VEL
LIN {X 0,Y 386.242,Z 449.488,A -85,B 0,C 180,E1 -11866.451,E2 -11866.451} C_VEL
LIN {X 0,Y 385.617,Z 459.938,A -85,B 0,C 180,E1 -11867.634,E2 -11867.634} C_VEL
LIN {X 0,Y 385.029,Z 469.511,A -85,B 0,C 180,E1 -11868.95,E2 -11868.95} C_VEL
LIN {X 0,Y 384.49,Z 477.457,A -85,B 0,C 180,E1 -11870.266,E2 -11870.266} C_VEL
LIN {X 0,Y 384.044,Z 485.248,A -85,B 0,C 180,E1 -11871.846,E2 -11871.846} C_VEL
LIN {X 0,Y 383.524,Z 492.519,A -85,B 0,C 180,E1 -11873.687,E2 -11873.687} C_VEL
LIN {X 0,Y 383.299,Z 497.365,A -85,B 0,C 180,E1 -11875.267,E2 -11875.267} C_VEL
LIN {X 0,Y 382.864,Z 501.132,A -85,B 0,C 180,E1 -11876.843,E2 -11876.843} C_VEL
LIN {X 0,Y 382.977,Z 503.008,A -85,B 0,C 180,E1 -11877.896,E2 -11877.896} C_VEL
LIN {X 0,Y 382.888,Z 504.518,A -85,B 0,C 180,E1 -11878.948,E2 -11878.948} C_VEL
LIN {X 0,Y 382.998,Z 505.595,A -85,B 0,C 180,E1 -11880,E2 -11880} C_VEL
LIN {X 0,Y 383.163,Z 506.482,A -85,B 0,C 180,E1 -11882.102,E2 -11882.102} C_VEL
LIN {X 0,Y 383.245,Z 506.356,A -85,B 0,C 180,E1 -11883.154,E2 -11883.154} C_VEL
LIN {X 0,Y 383.344,Z 505.791,A -85,B 0,C 180,E1 -11884.205,E2 -11884.205} C_VEL
LIN {X 0,Y 383.778,Z 503.445,A -85,B 0,C 180,E1 -11886.308,E2 -11886.308} C_VEL
LIN {X 0,Y 384.405,Z 500.507,A -85,B 0,C 180,E1 -11887.881,E2 -11887.881} C_VEL
LIN {X 0,Y 385.073,Z 495.658,A -85,B 0,C 180,E1 -11889.747,E2 -11889.747} C_VEL
LIN {X 0,Y 385.925,Z 489.38,A -85,B 0,C 180,E1 -11891.555,E2 -11891.555} C_VEL
LIN {X 0,Y 386.855,Z 482.395,A -85,B 0,C 180,E1 -11893.126,E2 -11893.126} C_VEL
LIN {X 0,Y 387.931,Z 473.693,A -85,B 0,C 180,E1 -11894.693,E2 -11894.693} C_VEL
LIN {X 0,Y 388.838,Z 465.124,A -85,B 0,C 180,E1 -11895.948,E2 -11895.948} C_VEL
LIN {X 0,Y 390.066,Z 453.815,A -85,B 0,C 180,E1 -11897.267,E2 -11897.267} C_VEL
LIN {X 0,Y 390.808,Z 444.953,A -85,B 0,C 180,E1 -11898.123,E2 -11898.123} C_VEL
LIN {X 0,Y 388.005,Z 435.982,A -85,B 0,C 180,E1 -11899.146,E2 -11899.146} C_VEL
LIN {X 0,Y 383.074,Z 423.975,A -85,B 0,C 180,E1 -11900.43,E2 -11900.43} C_VEL
LIN {X 0,Y 383.036,Z 423.775,A -85,B 0,C 180,E1 -11903.807,E2 -11903.807} C_VEL
LIN {X 0,Y 383.083,Z 423.766,A -85,B 0,C 180,E1 -11906.123,E2 -11906.123} C_VEL
LIN {X 0,Y 383.044,Z 423.772,A -85,B 0,C 180,E1 -11908.492,E2 -11908.492} C_VEL
LIN {X 0,Y 383.012,Z 423.776,A -85,B 0,C 180,E1 -11912.149,E2 -11912.149} C_VEL
LIN {X 0,Y 383.021,Z 423.776,A -85,B 0,C 180,E1 -11914.668,E2 -11914.668} C_VEL
LIN {X 0,Y 383.002,Z 423.776,A -85,B 0,C 180,E1 -11917.903,E2 -11917.903} C_VEL
LIN {X 0,Y 382.986,Z 423.774,A -85,B 0,C 180,E1 -11921.347,E2 -11921.347} C_VEL
LIN {X 0,Y 383.023,Z 423.777,A -85,B 0,C 180,E1 -11924.949,E2 -11924.949} C_VEL
LIN {X 0,Y 383.06,Z 424.082,A -85,B 0,C 180,E1 -11925.314,E2 -11925.314} C_VEL
LIN {X 0,Y 384.803,Z 432.309,A -85,B 0,C 180,E1 -11928.488,E2 -11928.488} C_VEL
LIN {X 0,Y 386.542,Z 441.551,A -85,B 0,C 180,E1 -11931.816,E2 -11931.816} C_VEL
LIN {X 0,Y 386.832,Z 445.279,A -85,B 0,C 180,E1 -11933.073,E2 -11933.073} C_VEL
LIN {X 0,Y 385.547,Z 457.723,A -85,B 0,C 180,E1 -11936.984,E2 -11936.984} C_VEL
LIN {X 0,Y 384.453,Z 470.784,A -85,B 0,C 180,E1 -11940.958,E2 -11940.958} C_VEL
LIN {X 0,Y 383.67,Z 482.668,A -85,B 0,C 180,E1 -11944.502,E2 -11944.502} C_VEL
LIN {X 0,Y 382.981,Z 494.169,A -85,B 0,C 180,E1 -11947.902,E2 -11947.902} C_VEL
LIN {X 0,Y 382.642,Z 502.438,A -85,B 0,C 180,E1 -11950.345,E2 -11950.345} C_VEL
LIN {X 0,Y 384.408,Z 515.474,A -85,B 0,C 180,E1 -11951.091,E2 -11951.091} C_VEL
LIN {X 0,Y 385.785,Z 534.61,A -85,B 0,C 180,E1 -11952.174,E2 -11952.174} C_VEL
LIN {X 0,Y 386.126,Z 547.111,A -85,B 0,C 180,E1 -11953.069,E2 -11953.069} C_VEL
LIN {X 0,Y 385.976,Z 553.397,A -85,B 0,C 180,E1 -11953.606,E2 -11953.606} C_VEL
LIN {X 0,Y 384.815,Z 565.139,A -85,B 0,C 180,E1 -11954.779,E2 -11954.779} C_VEL
LIN {X 0,Y 383.909,Z 574.84,A -85,B 0,C 180,E1 -11955.988,E2 -11955.988} C_VEL
LIN {X 0,Y 383.239,Z 583.387,A -85,B 0,C 180,E1 -11957.287,E2 -11957.287} C_VEL
LIN {X 0,Y 382.601,Z 591.915,A -85,B 0,C 180,E1 -11958.879,E2 -11958.879} C_VEL
LIN {X 0,Y 382.267,Z 598.84,A -85,B 0,C 180,E1 -11960.475,E2 -11960.475} C_VEL
LIN {X 0,Y 382.144,Z 604.41,A -85,B 0,C 180,E1 -11962.072,E2 -11962.072} C_VEL
LIN {X 0,Y 382.231,Z 608.798,A -85,B 0,C 180,E1 -11963.666,E2 -11963.666} C_VEL
LIN {X 0,Y 382.254,Z 611.129,A -85,B 0,C 180,E1 -11964.725,E2 -11964.725} C_VEL
LIN {X 0,Y 382.422,Z 612.985,A -85,B 0,C 180,E1 -11965.784,E2 -11965.784} C_VEL
LIN {X 0,Y 382.437,Z 614.385,A -85,B 0,C 180,E1 -11966.839,E2 -11966.839} C_VEL
LIN {X 0,Y 382.762,Z 616.006,A -85,B 0,C 180,E1 -11968.948,E2 -11968.948} C_VEL
LIN {X 0,Y 382.795,Z 616.146,A -85,B 0,C 180,E1 -11970,E2 -11970} C_VEL
LIN {X 0,Y 382.767,Z 615.867,A -85,B 0,C 180,E1 -11971.052,E2 -11971.052} C_VEL
LIN {X 0,Y 382.465,Z 614.061,A -85,B 0,C 180,E1 -11973.16,E2 -11973.16} C_VEL
LIN {X 0,Y 382.384,Z 611.566,A -85,B 0,C 180,E1 -11974.744,E2 -11974.744} C_VEL
LIN {X 0,Y 382.259,Z 608.028,A -85,B 0,C 180,E1 -11976.333,E2 -11976.333} C_VEL
LIN {X 0,Y 382.195,Z 603.376,A -85,B 0,C 180,E1 -11977.927,E2 -11977.927} C_VEL
LIN {X 0,Y 382.333,Z 596.357,A -85,B 0,C 180,E1 -11979.789,E2 -11979.789} C_VEL
LIN {X 0,Y 382.712,Z 588.757,A -85,B 0,C 180,E1 -11981.385,E2 -11981.385} C_VEL
LIN {X 0,Y 383.24,Z 581.048,A -85,B 0,C 180,E1 -11982.712,E2 -11982.712} C_VEL
LIN {X 0,Y 383.758,Z 572.616,A -85,B 0,C 180,E1 -11983.922,E2 -11983.922} C_VEL
LIN {X 0,Y 384.665,Z 562.718,A -85,B 0,C 180,E1 -11985.091,E2 -11985.091} C_VEL
LIN {X 0,Y 385.602,Z 551.701,A -85,B 0,C 180,E1 -11986.138,E2 -11986.138} C_VEL
LIN {X 0,Y 385.514,Z 544.93,A -85,B 0,C 180,E1 -11986.686,E2 -11986.686} C_VEL
LIN {X 0,Y 385.023,Z 532.219,A -85,B 0,C 180,E1 -11987.542,E2 -11987.542} C_VEL
LIN {X 0,Y 384.087,Z 518.973,A -85,B 0,C 180,E1 -11988.209,E2 -11988.209} C_VEL
LIN {X 0,Y 382.494,Z 504.29,A -85,B 0,C 180,E1 -11988.722,E2 -11988.722} C_VEL
LIN {X 0,Y 382.944,Z 492.715,A -85,B 0,C 180,E1 -11992.1,E2 -11992.1} C_VEL
LIN {X 0,Y 383.64,Z 479.063,A -85,B 0,C 180,E1 -11996.082,E2 -11996.082} C_VEL
LIN {X 0,Y 384.601,Z 465.186,A -85,B 0,C 180,E1 -12000.167,E2 -12000.167} C_VEL
LIN {X 0,Y 385.457,Z 453.17,A -85,B 0,C 180,E1 -12003.787,E2 -12003.787} C_VEL
LIN {X 0,Y 386.424,Z 443.155,A -85,B 0,C 180,E1 -12006.883,E2 -12006.883} C_VEL
LIN {X 0,Y 385.909,Z 438.418,A -85,B 0,C 180,E1 -12008.455,E2 -12008.455} C_VEL
LIN {X 0,Y 384.299,Z 429.954,A -85,B 0,C 180,E1 -12011.427,E2 -12011.427} C_VEL
LIN {X 0,Y 383.02,Z 423.777,A -85,B 0,C 180,E1 -12013.735,E2 -12013.735} C_VEL
LIN {X 0,Y 383.01,Z 423.781,A -85,B 0,C 180,E1 -12017.24,E2 -12017.24} C_VEL
LIN {X 0,Y 383.017,Z 423.777,A -85,B 0,C 180,E1 -12020.413,E2 -12020.413} C_VEL
LIN {X 0,Y 383.027,Z 423.776,A -85,B 0,C 180,E1 -12024.045,E2 -12024.045} C_VEL
LIN {X 0,Y 382.987,Z 423.776,A -85,B 0,C 180,E1 -12027.578,E2 -12027.578} C_VEL
LIN {X 0,Y 382.993,Z 423.78,A -85,B 0,C 180,E1 -12030.3,E2 -12030.3} C_VEL
LIN {X 0,Y 383.081,Z 423.769,A -85,B 0,C 180,E1 -12034.021,E2 -12034.021} C_VEL
LIN {X 0,Y 383.009,Z 423.773,A -85,B 0,C 180,E1 -12037.335,E2 -12037.335} C_VEL
LIN {X 0,Y 383.061,Z 423.768,A -85,B 0,C 180,E1 -12040.716,E2 -12040.716} C_VEL
LIN {X 0,Y 383.082,Z 423.769,A -85,B 0,C 180,E1 -12044.027,E2 -12044.027} C_VEL
LIN {X 0,Y 383.142,Z 423.757,A -85,B 0,C 180,E1 -12047.284,E2 -12047.284} C_VEL
LIN {X 0,Y 383.149,Z 423.758,A -85,B 0,C 180,E1 -12050.498,E2 -12050.498} C_VEL
LIN {X 0,Y 383.277,Z 423.742,A -85,B 0,C 180,E1 -12053.684,E2 -12053.684} C_VEL
LIN {X 0,Y 383.39,Z 423.73,A -85,B 0,C 180,E1 -12057.899,E2 -12057.899} C_VEL
LIN {X 0,Y 383.521,Z 423.715,A -85,B 0,C 180,E1 -12060,E2 -12060} C_VEL
LIN {X 0,Y 383.248,Z 423.743,A -85,B 0,C 180,E1 -12063.154,E2 -12063.154} C_VEL
LIN {X 0,Y 383.27,Z 423.741,A -85,B 0,C 180,E1 -12066.648,E2 -12066.648} C_VEL
LIN {X 0,Y 383.261,Z 423.744,A -85,B 0,C 180,E1 -12068.436,E2 -12068.436} C_VEL
LIN {X 0,Y 383.1,Z 423.765,A -85,B 0,C 180,E1 -12071.642,E2 -12071.642} C_VEL
LIN {X 0,Y 383.112,Z 423.76,A -85,B 0,C 180,E1 -12074.882,E2 -12074.882} C_VEL
LIN {X 0,Y 383.091,Z 423.767,A -85,B 0,C 180,E1 -12078.172,E2 -12078.172} C_VEL
LIN {X 0,Y 382.995,Z 423.777,A -85,B 0,C 180,E1 -12081.531,E2 -12081.531} C_VEL
LIN {X 0,Y 383.054,Z 423.767,A -85,B 0,C 180,E1 -12084.96,E2 -12084.96} C_VEL
LIN {X 0,Y 383.019,Z 423.773,A -85,B 0,C 180,E1 -12088.495,E2 -12088.495} C_VEL
LIN {X 0,Y 383.011,Z 423.777,A -85,B 0,C 180,E1 -12092.15,E2 -12092.15} C_VEL
LIN {X 0,Y 383.02,Z 423.772,A -85,B 0,C 180,E1 -12094.668,E2 -12094.668} C_VEL
LIN {X 0,Y 383.003,Z 423.78,A -85,B 0,C 180,E1 -12097.904,E2 -12097.904} C_VEL
LIN {X 0,Y 382.987,Z 423.777,A -85,B 0,C 180,E1 -12101.347,E2 -12101.347} C_VEL
LIN {X 0,Y 383.001,Z 423.776,A -85,B 0,C 180,E1 -12104.304,E2 -12104.304} C_VEL
LIN {X 0,Y 383.012,Z 423.774,A -85,B 0,C 180,E1 -12107.241,E2 -12107.241} C_VEL
LIN {X 0,Y 383.018,Z 423.773,A -85,B 0,C 180,E1 -12110.414,E2 -12110.414} C_VEL
LIN {X 0,Y 383.029,Z 423.774,A -85,B 0,C 180,E1 -12114.045,E2 -12114.045} C_VEL
LIN {X 0,Y 383.04,Z 423.774,A -85,B 0,C 180,E1 -12117.853,E2 -12117.853} C_VEL
LIN {X 0,Y 383.067,Z 423.771,A -85,B 0,C 180,E1 -12121.721,E2 -12121.721} C_VEL
LIN {X 0,Y 383.056,Z 423.768,A -85,B 0,C 180,E1 -12125.04,E2 -12125.04} C_VEL
LIN {X 0,Y 382.997,Z 423.775,A -85,B 0,C 180,E1 -12128.469,E2 -12128.469} C_VEL
LIN {X 0,Y 383.093,Z 423.767,A -85,B 0,C 180,E1 -12131.828,E2 -12131.828} C_VEL
LIN {X 0,Y 383.111,Z 423.868,A -85,B 0,C 180,E1 -12135.305,E2 -12135.305} C_VEL
LIN {X 0,Y 386.708,Z 435.545,A -85,B 0,C 180,E1 -12136.241,E2 -12136.241} C_VEL
LIN {X 0,Y 388.315,Z 441.392,A -85,B 0,C 180,E1 -12136.792,E2 -12136.792} C_VEL
LIN {X 0,Y 387.662,Z 452.625,A -85,B 0,C 180,E1 -12137.834,E2 -12137.834} C_VEL
LIN {X 0,Y 386.866,Z 462.606,A -85,B 0,C 180,E1 -12138.984,E2 -12138.984} C_VEL
LIN {X 0,Y 386.048,Z 471.864,A -85,B 0,C 180,E1 -12140.306,E2 -12140.306} C_VEL
LIN {X 0,Y 385.322,Z 480.645,A -85,B 0,C 180,E1 -12141.874,E2 -12141.874} C_VEL
LIN {X 0,Y 384.593,Z 487.736,A -85,B 0,C 180,E1 -12143.442,E2 -12143.442} C_VEL
LIN {X 0,Y 383.992,Z 494.202,A -85,B 0,C 180,E1 -12145.276,E2 -12145.276} C_VEL
LIN {X 0,Y 383.585,Z 498.477,A -85,B 0,C 180,E1 -12146.849,E2 -12146.849} C_VEL
LIN {X 0,Y 383.339,Z 500.743,A -85,B 0,C 180,E1 -12147.899,E2 -12147.899} C_VEL
LIN {X 0,Y 383.162,Z 502.591,A -85,B 0,C 180,E1 -12148.949,E2 -12148.949} C_VEL
LIN {X 0,Y 383.076,Z 504,A -85,B 0,C 180,E1 -12150,E2 -12150} C_VEL
LIN {X 0,Y 382.958,Z 505.627,A -85,B 0,C 180,E1 -12152.104,E2 -12152.104} C_VEL
LIN {X 0,Y 382.836,Z 505.903,A -85,B 0,C 180,E1 -12153.157,E2 -12153.157} C_VEL
LIN {X 0,Y 382.915,Z 505.755,A -85,B 0,C 180,E1 -12154.21,E2 -12154.21} C_VEL
LIN {X 0,Y 383.325,Z 504.259,A -85,B 0,C 180,E1 -12156.316,E2 -12156.316} C_VEL
LIN {X 0,Y 383.444,Z 502.964,A -85,B 0,C 180,E1 -12157.372,E2 -12157.372} C_VEL
LIN {X 0,Y 383.779,Z 500.195,A -85,B 0,C 180,E1 -12158.955,E2 -12158.955} C_VEL
LIN {X 0,Y 384.33,Z 496.403,A -85,B 0,C 180,E1 -12160.537,E2 -12160.537} C_VEL
LIN {X 0,Y 384.879,Z 491.509,A -85,B 0,C 180,E1 -12162.122,E2 -12162.122} C_VEL
LIN {X 0,Y 385.48,Z 485.333,A -85,B 0,C 180,E1 -12163.711,E2 -12163.711} C_VEL
LIN {X 0,Y 386.173,Z 478.734,A -85,B 0,C 180,E1 -12165.082,E2 -12165.082} C_VEL
LIN {X 0,Y 387.135,Z 469.586,A -85,B 0,C 180,E1 -12166.614,E2 -12166.614} C_VEL
LIN {X 0,Y 387.957,Z 459.845,A -85,B 0,C 180,E1 -12167.937,E2 -12167.937} C_VEL
LIN {X 0,Y 388.886,Z 448.888,A -85,B 0,C 180,E1 -12169.113,E2 -12169.113} C_VEL
LIN {X 0,Y 389.189,Z 443.945,A -85,B 0,C 180,E1 -12169.564,E2 -12169.564} C_VEL
LIN {X 0,Y 387.778,Z 438.104,A -85,B 0,C 180,E1 -12170.143,E2 -12170.143} C_VEL
LIN {X 0,Y 384.197,Z 427.501,A -85,B 0,C 180,E1 -12171.103,E2 -12171.103} C_VEL
